// TwinCAT 3 PLC project PLC
// ProgramVersion: 3.1.4023.0
// libraries:
//   Tc2_Standard, * (Beckhoff Automation GmbH)
//   Tc2_System, * (Beckhoff Automation GmbH)
//   Tc3_Module, * (Beckhoff Automation GmbH)
// project tree:
//   / PlcTask.TcTTO
//   POUs/ MAIN.TcPOU
//   DUTs/IO/PDOs/ InfoData_6F19DB2B.TcDUT, YVR_Inputs_4719D0DB.TcDUT, YVR_Outputs_31F2CBB3.TcDUT, WcState_9091E0EB.TcDUT, InfoData_BEF6B88E.TcDUT, FB_Inputs_F0F03BDD.TcDUT, InfoData_A7436BC6.TcDUT, APS_Inputs_4719D0DB.TcDUT, APS_Diagdata_CE5B986F.TcDUT, APS_Comm_Inputs_388FE28E.TcDUT, APS_Outputs_31F2CBB3.TcDUT, APS_Comm_Outputs_082002A4.TcDUT, InfoData_E68C61CD.TcDUT, WcState_0B2B16F9.TcDUT, InfoData_2A97D6CF.TcDUT, Inputs_25A0042B.TcDUT, Outputs_2397A10E.TcDUT
//   DUTs/IO/Boxes/ EK1100_1FC0878B.TcDUT, EK1122_1FC0878B.TcDUT, APS1003_C6D7567B.TcDUT, APS1003_A49C5437.TcDUT, APS4322_7CC84994.TcDUT, APS4322_A49C5437.TcDUT
//   DUTs/IO/Devices/ SyncUnitTask_2D604ED5.TcDUT, SyncUnitTasks_6FEB8257.TcDUT, SyncUnits_99E584AF.TcDUT
//   DUTs/IO/Topology/ Beckhoff_APS1xxxEK1122_94631AF6.TcDUT, Beckhoff_APS1xxx_5C0D85AF.TcDUT, Beckhoff_APS4xxxEK1122_0B49C1F2.TcDUT, Beckhoff_APS4xxx_9BEEA20F.TcDUT, EtherCAT_Master_APSxxxx_214E63DA.TcDUT
//   DUTs/IO/Base/ EtcSlaveBase_82538BE2.TcDUT, EtcSlaveBase_82538BE2.TcDUT, EtcSlaveBase_82538BE2.TcDUT, EtcSlaveTerminalBase_947E5A46.TcDUT, EtcSlaveBoxBase_77A0E4A7.TcDUT, EtcSlaveEndTerminalBase_866C7F0C.TcDUT, InputBase_8311D824.TcDUT, OutputBase_10CEE7DE.TcDUT, EtcMasterBase_62654B43.TcDUT
//   GVLs/ GVL_iXlinker.TcGVL
// real-time tasks:
//   TASK PlcTask: cycle T#10ms, priority 20, ADS port 350
// I/O:
//   DEVICE EtherCAT_Master_APSxxxx, AmsNetId 172.20.30.238.3.1
//     Beckhoff APS1xxx [EK1100 EtherCAT Coupler (2A E-Bus)]
//       Beckhoff APS1xxxEK1122 [EK1122 2 port EtherCAT junction]
//         Beckhoff APS1xxxsub EK1100 [EK1100 EtherCAT Coupler (2A E-Bus)]
//         A_0001(APS1003-7000-0016) [APS1003-7000 Drive]
//       A_0002(APS1003-5000-0016) [APS1003-5000 Feedback]
//     Beckhoff APS4xxx [EK1100 EtherCAT Coupler (2A E-Bus)]
//       Beckhoff APS4xxxEK1122 [EK1122 2 port EtherCAT junction]
//         Beckhoff APS4xxxsub EK1100 [EK1100 EtherCAT Coupler (2A E-Bus)]
//         A_0001(APS4322-7000-0017) [APS4322-7000 Drive]
//       A_0002(APS4322-5000-0017) [APS4322-5000 Feedback]
// variable links:
//   PLC/PLC Instance <-> EtherCAT Master APSxxxx/Beckhoff APS1xxx
//     PlcTask Inputs/GVL_iXlinker.EtherCAT_Master_APSxxxx.Beckhoff_APS1xxx.InfoData.State <-> InfoData/State
//   PLC/PLC Instance <-> EtherCAT Master APSxxxx/Beckhoff APS1xxx/Beckhoff APS1xxxEK1122
//     PlcTask Inputs/GVL_iXlinker.EtherCAT_Master_APSxxxx.Beckhoff_APS1xxx.Beckhoff_APS1xxxEK1122.InfoData.State <-> InfoData/State
//   PLC/PLC Instance <-> EtherCAT Master APSxxxx/Beckhoff APS1xxx/Beckhoff APS1xxxEK1122/Beckhoff APS1xxxsub EK1100
//     PlcTask Inputs/GVL_iXlinker.EtherCAT_Master_APSxxxx.Beckhoff_APS1xxx.Beckhoff_APS1xxxEK1122.Beckhoff_APS1xxxsub_EK1100.InfoData.State <-> InfoData/State
//   PLC/PLC Instance <-> EtherCAT Master APSxxxx/Beckhoff APS1xxx/Beckhoff APS1xxxEK1122/A_0001(APS1003-7000-0016)
//     PlcTask Inputs/GVL_iXlinker.EtherCAT_Master_APSxxxx.Beckhoff_APS1xxx.Beckhoff_APS1xxxEK1122.A_0001_APS1003_7000_0016.YVR_Inputs.StatusWord <-> YVR Inputs/StatusWord
//     PlcTask Inputs/GVL_iXlinker.EtherCAT_Master_APSxxxx.Beckhoff_APS1xxx.Beckhoff_APS1xxxEK1122.A_0001_APS1003_7000_0016.YVR_Inputs.Current_D_0X0 <-> YVR Inputs/Current D 0X0
//     PlcTask Inputs/GVL_iXlinker.EtherCAT_Master_APSxxxx.Beckhoff_APS1xxx.Beckhoff_APS1xxxEK1122.A_0001_APS1003_7000_0016.YVR_Inputs.Current_D_0X1 <-> YVR Inputs/Current D 0X1
//     PlcTask Inputs/GVL_iXlinker.EtherCAT_Master_APSxxxx.Beckhoff_APS1xxx.Beckhoff_APS1xxxEK1122.A_0001_APS1003_7000_0016.YVR_Inputs.Current_D_0X2 <-> YVR Inputs/Current D 0X2
//     PlcTask Inputs/GVL_iXlinker.EtherCAT_Master_APSxxxx.Beckhoff_APS1xxx.Beckhoff_APS1xxxEK1122.A_0001_APS1003_7000_0016.YVR_Inputs.Current_D_1X0 <-> YVR Inputs/Current D 1X0
//     PlcTask Inputs/GVL_iXlinker.EtherCAT_Master_APSxxxx.Beckhoff_APS1xxx.Beckhoff_APS1xxxEK1122.A_0001_APS1003_7000_0016.YVR_Inputs.Current_D_1X1 <-> YVR Inputs/Current D 1X1
//     PlcTask Inputs/GVL_iXlinker.EtherCAT_Master_APSxxxx.Beckhoff_APS1xxx.Beckhoff_APS1xxxEK1122.A_0001_APS1003_7000_0016.YVR_Inputs.Current_D_1X2 <-> YVR Inputs/Current D 1X2
//     PlcTask Inputs/GVL_iXlinker.EtherCAT_Master_APSxxxx.Beckhoff_APS1xxx.Beckhoff_APS1xxxEK1122.A_0001_APS1003_7000_0016.YVR_Inputs.Current_D_2X0 <-> YVR Inputs/Current D 2X0
//     PlcTask Inputs/GVL_iXlinker.EtherCAT_Master_APSxxxx.Beckhoff_APS1xxx.Beckhoff_APS1xxxEK1122.A_0001_APS1003_7000_0016.YVR_Inputs.Current_D_2X1 <-> YVR Inputs/Current D 2X1
//     PlcTask Inputs/GVL_iXlinker.EtherCAT_Master_APSxxxx.Beckhoff_APS1xxx.Beckhoff_APS1xxxEK1122.A_0001_APS1003_7000_0016.YVR_Inputs.Current_D_2X2 <-> YVR Inputs/Current D 2X2
//     PlcTask Inputs/GVL_iXlinker.EtherCAT_Master_APSxxxx.Beckhoff_APS1xxx.Beckhoff_APS1xxxEK1122.A_0001_APS1003_7000_0016.YVR_Inputs.Current_D_3X0 <-> YVR Inputs/Current D 3X0
//     PlcTask Inputs/GVL_iXlinker.EtherCAT_Master_APSxxxx.Beckhoff_APS1xxx.Beckhoff_APS1xxxEK1122.A_0001_APS1003_7000_0016.YVR_Inputs.Current_D_3X1 <-> YVR Inputs/Current D 3X1
//     PlcTask Inputs/GVL_iXlinker.EtherCAT_Master_APSxxxx.Beckhoff_APS1xxx.Beckhoff_APS1xxxEK1122.A_0001_APS1003_7000_0016.YVR_Inputs.Current_D_3X2 <-> YVR Inputs/Current D 3X2
//     PlcTask Inputs/GVL_iXlinker.EtherCAT_Master_APSxxxx.Beckhoff_APS1xxx.Beckhoff_APS1xxxEK1122.A_0001_APS1003_7000_0016.YVR_Inputs.Current_D_0Y0 <-> YVR Inputs/Current D 0Y0
//     PlcTask Inputs/GVL_iXlinker.EtherCAT_Master_APSxxxx.Beckhoff_APS1xxx.Beckhoff_APS1xxxEK1122.A_0001_APS1003_7000_0016.YVR_Inputs.Current_D_0Y1 <-> YVR Inputs/Current D 0Y1
//     PlcTask Inputs/GVL_iXlinker.EtherCAT_Master_APSxxxx.Beckhoff_APS1xxx.Beckhoff_APS1xxxEK1122.A_0001_APS1003_7000_0016.YVR_Inputs.Current_D_0Y2 <-> YVR Inputs/Current D 0Y2
//     PlcTask Inputs/GVL_iXlinker.EtherCAT_Master_APSxxxx.Beckhoff_APS1xxx.Beckhoff_APS1xxxEK1122.A_0001_APS1003_7000_0016.YVR_Inputs.Current_D_1Y0 <-> YVR Inputs/Current D 1Y0
//     PlcTask Inputs/GVL_iXlinker.EtherCAT_Master_APSxxxx.Beckhoff_APS1xxx.Beckhoff_APS1xxxEK1122.A_0001_APS1003_7000_0016.YVR_Inputs.Current_D_1Y1 <-> YVR Inputs/Current D 1Y1
//     PlcTask Inputs/GVL_iXlinker.EtherCAT_Master_APSxxxx.Beckhoff_APS1xxx.Beckhoff_APS1xxxEK1122.A_0001_APS1003_7000_0016.YVR_Inputs.Current_D_1Y2 <-> YVR Inputs/Current D 1Y2
//     PlcTask Inputs/GVL_iXlinker.EtherCAT_Master_APSxxxx.Beckhoff_APS1xxx.Beckhoff_APS1xxxEK1122.A_0001_APS1003_7000_0016.YVR_Inputs.Current_D_2Y0 <-> YVR Inputs/Current D 2Y0
//     PlcTask Inputs/GVL_iXlinker.EtherCAT_Master_APSxxxx.Beckhoff_APS1xxx.Beckhoff_APS1xxxEK1122.A_0001_APS1003_7000_0016.YVR_Inputs.Current_D_2Y1 <-> YVR Inputs/Current D 2Y1
//     PlcTask Inputs/GVL_iXlinker.EtherCAT_Master_APSxxxx.Beckhoff_APS1xxx.Beckhoff_APS1xxxEK1122.A_0001_APS1003_7000_0016.YVR_Inputs.Current_D_2Y2 <-> YVR Inputs/Current D 2Y2
//     PlcTask Inputs/GVL_iXlinker.EtherCAT_Master_APSxxxx.Beckhoff_APS1xxx.Beckhoff_APS1xxxEK1122.A_0001_APS1003_7000_0016.YVR_Inputs.Current_D_3Y0 <-> YVR Inputs/Current D 3Y0
//     PlcTask Inputs/GVL_iXlinker.EtherCAT_Master_APSxxxx.Beckhoff_APS1xxx.Beckhoff_APS1xxxEK1122.A_0001_APS1003_7000_0016.YVR_Inputs.Current_D_3Y1 <-> YVR Inputs/Current D 3Y1
//     PlcTask Inputs/GVL_iXlinker.EtherCAT_Master_APSxxxx.Beckhoff_APS1xxx.Beckhoff_APS1xxxEK1122.A_0001_APS1003_7000_0016.YVR_Inputs.Current_D_3Y2 <-> YVR Inputs/Current D 3Y2
//     PlcTask Inputs/GVL_iXlinker.EtherCAT_Master_APSxxxx.Beckhoff_APS1xxx.Beckhoff_APS1xxxEK1122.A_0001_APS1003_7000_0016.YVR_Inputs.Current_Q_0X0 <-> YVR Inputs/Current Q 0X0
//     PlcTask Inputs/GVL_iXlinker.EtherCAT_Master_APSxxxx.Beckhoff_APS1xxx.Beckhoff_APS1xxxEK1122.A_0001_APS1003_7000_0016.YVR_Inputs.Current_Q_0X1 <-> YVR Inputs/Current Q 0X1
//     PlcTask Inputs/GVL_iXlinker.EtherCAT_Master_APSxxxx.Beckhoff_APS1xxx.Beckhoff_APS1xxxEK1122.A_0001_APS1003_7000_0016.YVR_Inputs.Current_Q_0X2 <-> YVR Inputs/Current Q 0X2
//     PlcTask Inputs/GVL_iXlinker.EtherCAT_Master_APSxxxx.Beckhoff_APS1xxx.Beckhoff_APS1xxxEK1122.A_0001_APS1003_7000_0016.YVR_Inputs.Current_Q_1X0 <-> YVR Inputs/Current Q 1X0
//     PlcTask Inputs/GVL_iXlinker.EtherCAT_Master_APSxxxx.Beckhoff_APS1xxx.Beckhoff_APS1xxxEK1122.A_0001_APS1003_7000_0016.YVR_Inputs.Current_Q_1X1 <-> YVR Inputs/Current Q 1X1
//     PlcTask Inputs/GVL_iXlinker.EtherCAT_Master_APSxxxx.Beckhoff_APS1xxx.Beckhoff_APS1xxxEK1122.A_0001_APS1003_7000_0016.YVR_Inputs.Current_Q_1X2 <-> YVR Inputs/Current Q 1X2
//     PlcTask Inputs/GVL_iXlinker.EtherCAT_Master_APSxxxx.Beckhoff_APS1xxx.Beckhoff_APS1xxxEK1122.A_0001_APS1003_7000_0016.YVR_Inputs.Current_Q_2X0 <-> YVR Inputs/Current Q 2X0
//     PlcTask Inputs/GVL_iXlinker.EtherCAT_Master_APSxxxx.Beckhoff_APS1xxx.Beckhoff_APS1xxxEK1122.A_0001_APS1003_7000_0016.YVR_Inputs.Current_Q_2X1 <-> YVR Inputs/Current Q 2X1
//     PlcTask Inputs/GVL_iXlinker.EtherCAT_Master_APSxxxx.Beckhoff_APS1xxx.Beckhoff_APS1xxxEK1122.A_0001_APS1003_7000_0016.YVR_Inputs.Current_Q_2X2 <-> YVR Inputs/Current Q 2X2
//     PlcTask Inputs/GVL_iXlinker.EtherCAT_Master_APSxxxx.Beckhoff_APS1xxx.Beckhoff_APS1xxxEK1122.A_0001_APS1003_7000_0016.YVR_Inputs.Current_Q_3X0 <-> YVR Inputs/Current Q 3X0
//     PlcTask Inputs/GVL_iXlinker.EtherCAT_Master_APSxxxx.Beckhoff_APS1xxx.Beckhoff_APS1xxxEK1122.A_0001_APS1003_7000_0016.YVR_Inputs.Current_Q_3X1 <-> YVR Inputs/Current Q 3X1
//     PlcTask Inputs/GVL_iXlinker.EtherCAT_Master_APSxxxx.Beckhoff_APS1xxx.Beckhoff_APS1xxxEK1122.A_0001_APS1003_7000_0016.YVR_Inputs.Current_Q_3X2 <-> YVR Inputs/Current Q 3X2
//     PlcTask Inputs/GVL_iXlinker.EtherCAT_Master_APSxxxx.Beckhoff_APS1xxx.Beckhoff_APS1xxxEK1122.A_0001_APS1003_7000_0016.YVR_Inputs.Current_Q_0Y0 <-> YVR Inputs/Current Q 0Y0
//     PlcTask Inputs/GVL_iXlinker.EtherCAT_Master_APSxxxx.Beckhoff_APS1xxx.Beckhoff_APS1xxxEK1122.A_0001_APS1003_7000_0016.YVR_Inputs.Current_Q_0Y1 <-> YVR Inputs/Current Q 0Y1
//     PlcTask Inputs/GVL_iXlinker.EtherCAT_Master_APSxxxx.Beckhoff_APS1xxx.Beckhoff_APS1xxxEK1122.A_0001_APS1003_7000_0016.YVR_Inputs.Current_Q_0Y2 <-> YVR Inputs/Current Q 0Y2
//     PlcTask Inputs/GVL_iXlinker.EtherCAT_Master_APSxxxx.Beckhoff_APS1xxx.Beckhoff_APS1xxxEK1122.A_0001_APS1003_7000_0016.YVR_Inputs.Current_Q_1Y0 <-> YVR Inputs/Current Q 1Y0
//     PlcTask Inputs/GVL_iXlinker.EtherCAT_Master_APSxxxx.Beckhoff_APS1xxx.Beckhoff_APS1xxxEK1122.A_0001_APS1003_7000_0016.YVR_Inputs.Current_Q_1Y1 <-> YVR Inputs/Current Q 1Y1
//     PlcTask Inputs/GVL_iXlinker.EtherCAT_Master_APSxxxx.Beckhoff_APS1xxx.Beckhoff_APS1xxxEK1122.A_0001_APS1003_7000_0016.YVR_Inputs.Current_Q_1Y2 <-> YVR Inputs/Current Q 1Y2
//     PlcTask Inputs/GVL_iXlinker.EtherCAT_Master_APSxxxx.Beckhoff_APS1xxx.Beckhoff_APS1xxxEK1122.A_0001_APS1003_7000_0016.YVR_Inputs.Current_Q_2Y0 <-> YVR Inputs/Current Q 2Y0
//     PlcTask Inputs/GVL_iXlinker.EtherCAT_Master_APSxxxx.Beckhoff_APS1xxx.Beckhoff_APS1xxxEK1122.A_0001_APS1003_7000_0016.YVR_Inputs.Current_Q_2Y1 <-> YVR Inputs/Current Q 2Y1
//     PlcTask Inputs/GVL_iXlinker.EtherCAT_Master_APSxxxx.Beckhoff_APS1xxx.Beckhoff_APS1xxxEK1122.A_0001_APS1003_7000_0016.YVR_Inputs.Current_Q_2Y2 <-> YVR Inputs/Current Q 2Y2
//     PlcTask Inputs/GVL_iXlinker.EtherCAT_Master_APSxxxx.Beckhoff_APS1xxx.Beckhoff_APS1xxxEK1122.A_0001_APS1003_7000_0016.YVR_Inputs.Current_Q_3Y0 <-> YVR Inputs/Current Q 3Y0
//     PlcTask Inputs/GVL_iXlinker.EtherCAT_Master_APSxxxx.Beckhoff_APS1xxx.Beckhoff_APS1xxxEK1122.A_0001_APS1003_7000_0016.YVR_Inputs.Current_Q_3Y1 <-> YVR Inputs/Current Q 3Y1
//     PlcTask Inputs/GVL_iXlinker.EtherCAT_Master_APSxxxx.Beckhoff_APS1xxx.Beckhoff_APS1xxxEK1122.A_0001_APS1003_7000_0016.YVR_Inputs.Current_Q_3Y2 <-> YVR Inputs/Current Q 3Y2
//     PlcTask Outputs/GVL_iXlinker.EtherCAT_Master_APSxxxx.Beckhoff_APS1xxx.Beckhoff_APS1xxxEK1122.A_0001_APS1003_7000_0016.YVR_Outputs.ControlWord <-> YVR Outputs/ControlWord
//     PlcTask Outputs/GVL_iXlinker.EtherCAT_Master_APSxxxx.Beckhoff_APS1xxx.Beckhoff_APS1xxxEK1122.A_0001_APS1003_7000_0016.YVR_Outputs.Current_D_0X0 <-> YVR Outputs/Current D 0X0
//     PlcTask Outputs/GVL_iXlinker.EtherCAT_Master_APSxxxx.Beckhoff_APS1xxx.Beckhoff_APS1xxxEK1122.A_0001_APS1003_7000_0016.YVR_Outputs.Current_D_0X1 <-> YVR Outputs/Current D 0X1
//     PlcTask Outputs/GVL_iXlinker.EtherCAT_Master_APSxxxx.Beckhoff_APS1xxx.Beckhoff_APS1xxxEK1122.A_0001_APS1003_7000_0016.YVR_Outputs.Current_D_0X2 <-> YVR Outputs/Current D 0X2
//     PlcTask Outputs/GVL_iXlinker.EtherCAT_Master_APSxxxx.Beckhoff_APS1xxx.Beckhoff_APS1xxxEK1122.A_0001_APS1003_7000_0016.YVR_Outputs.Current_D_1X0 <-> YVR Outputs/Current D 1X0
//     PlcTask Outputs/GVL_iXlinker.EtherCAT_Master_APSxxxx.Beckhoff_APS1xxx.Beckhoff_APS1xxxEK1122.A_0001_APS1003_7000_0016.YVR_Outputs.Current_D_1X1 <-> YVR Outputs/Current D 1X1
//     PlcTask Outputs/GVL_iXlinker.EtherCAT_Master_APSxxxx.Beckhoff_APS1xxx.Beckhoff_APS1xxxEK1122.A_0001_APS1003_7000_0016.YVR_Outputs.Current_D_1X2 <-> YVR Outputs/Current D 1X2
//     PlcTask Outputs/GVL_iXlinker.EtherCAT_Master_APSxxxx.Beckhoff_APS1xxx.Beckhoff_APS1xxxEK1122.A_0001_APS1003_7000_0016.YVR_Outputs.Current_D_2X0 <-> YVR Outputs/Current D 2X0
//     PlcTask Outputs/GVL_iXlinker.EtherCAT_Master_APSxxxx.Beckhoff_APS1xxx.Beckhoff_APS1xxxEK1122.A_0001_APS1003_7000_0016.YVR_Outputs.Current_D_2X1 <-> YVR Outputs/Current D 2X1
//     PlcTask Outputs/GVL_iXlinker.EtherCAT_Master_APSxxxx.Beckhoff_APS1xxx.Beckhoff_APS1xxxEK1122.A_0001_APS1003_7000_0016.YVR_Outputs.Current_D_2X2 <-> YVR Outputs/Current D 2X2
//     PlcTask Outputs/GVL_iXlinker.EtherCAT_Master_APSxxxx.Beckhoff_APS1xxx.Beckhoff_APS1xxxEK1122.A_0001_APS1003_7000_0016.YVR_Outputs.Current_D_3X0 <-> YVR Outputs/Current D 3X0
//     PlcTask Outputs/GVL_iXlinker.EtherCAT_Master_APSxxxx.Beckhoff_APS1xxx.Beckhoff_APS1xxxEK1122.A_0001_APS1003_7000_0016.YVR_Outputs.Current_D_3X1 <-> YVR Outputs/Current D 3X1
//     PlcTask Outputs/GVL_iXlinker.EtherCAT_Master_APSxxxx.Beckhoff_APS1xxx.Beckhoff_APS1xxxEK1122.A_0001_APS1003_7000_0016.YVR_Outputs.Current_D_3X2 <-> YVR Outputs/Current D 3X2
//     PlcTask Outputs/GVL_iXlinker.EtherCAT_Master_APSxxxx.Beckhoff_APS1xxx.Beckhoff_APS1xxxEK1122.A_0001_APS1003_7000_0016.YVR_Outputs.Current_D_0Y0 <-> YVR Outputs/Current D 0Y0
//     PlcTask Outputs/GVL_iXlinker.EtherCAT_Master_APSxxxx.Beckhoff_APS1xxx.Beckhoff_APS1xxxEK1122.A_0001_APS1003_7000_0016.YVR_Outputs.Current_D_0Y1 <-> YVR Outputs/Current D 0Y1
//     PlcTask Outputs/GVL_iXlinker.EtherCAT_Master_APSxxxx.Beckhoff_APS1xxx.Beckhoff_APS1xxxEK1122.A_0001_APS1003_7000_0016.YVR_Outputs.Current_D_0Y2 <-> YVR Outputs/Current D 0Y2
//     PlcTask Outputs/GVL_iXlinker.EtherCAT_Master_APSxxxx.Beckhoff_APS1xxx.Beckhoff_APS1xxxEK1122.A_0001_APS1003_7000_0016.YVR_Outputs.Current_D_1Y0 <-> YVR Outputs/Current D 1Y0
//     PlcTask Outputs/GVL_iXlinker.EtherCAT_Master_APSxxxx.Beckhoff_APS1xxx.Beckhoff_APS1xxxEK1122.A_0001_APS1003_7000_0016.YVR_Outputs.Current_D_1Y1 <-> YVR Outputs/Current D 1Y1
//     PlcTask Outputs/GVL_iXlinker.EtherCAT_Master_APSxxxx.Beckhoff_APS1xxx.Beckhoff_APS1xxxEK1122.A_0001_APS1003_7000_0016.YVR_Outputs.Current_D_1Y2 <-> YVR Outputs/Current D 1Y2
//     PlcTask Outputs/GVL_iXlinker.EtherCAT_Master_APSxxxx.Beckhoff_APS1xxx.Beckhoff_APS1xxxEK1122.A_0001_APS1003_7000_0016.YVR_Outputs.Current_D_2Y0 <-> YVR Outputs/Current D 2Y0
//     PlcTask Outputs/GVL_iXlinker.EtherCAT_Master_APSxxxx.Beckhoff_APS1xxx.Beckhoff_APS1xxxEK1122.A_0001_APS1003_7000_0016.YVR_Outputs.Current_D_2Y1 <-> YVR Outputs/Current D 2Y1
//     PlcTask Outputs/GVL_iXlinker.EtherCAT_Master_APSxxxx.Beckhoff_APS1xxx.Beckhoff_APS1xxxEK1122.A_0001_APS1003_7000_0016.YVR_Outputs.Current_D_2Y2 <-> YVR Outputs/Current D 2Y2
//     PlcTask Outputs/GVL_iXlinker.EtherCAT_Master_APSxxxx.Beckhoff_APS1xxx.Beckhoff_APS1xxxEK1122.A_0001_APS1003_7000_0016.YVR_Outputs.Current_D_3Y0 <-> YVR Outputs/Current D 3Y0
//     PlcTask Outputs/GVL_iXlinker.EtherCAT_Master_APSxxxx.Beckhoff_APS1xxx.Beckhoff_APS1xxxEK1122.A_0001_APS1003_7000_0016.YVR_Outputs.Current_D_3Y1 <-> YVR Outputs/Current D 3Y1
//     PlcTask Outputs/GVL_iXlinker.EtherCAT_Master_APSxxxx.Beckhoff_APS1xxx.Beckhoff_APS1xxxEK1122.A_0001_APS1003_7000_0016.YVR_Outputs.Current_D_3Y2 <-> YVR Outputs/Current D 3Y2
//     PlcTask Outputs/GVL_iXlinker.EtherCAT_Master_APSxxxx.Beckhoff_APS1xxx.Beckhoff_APS1xxxEK1122.A_0001_APS1003_7000_0016.YVR_Outputs.Current_Q_0X0 <-> YVR Outputs/Current Q 0X0
//     PlcTask Outputs/GVL_iXlinker.EtherCAT_Master_APSxxxx.Beckhoff_APS1xxx.Beckhoff_APS1xxxEK1122.A_0001_APS1003_7000_0016.YVR_Outputs.Current_Q_0X1 <-> YVR Outputs/Current Q 0X1
//     PlcTask Outputs/GVL_iXlinker.EtherCAT_Master_APSxxxx.Beckhoff_APS1xxx.Beckhoff_APS1xxxEK1122.A_0001_APS1003_7000_0016.YVR_Outputs.Current_Q_0X2 <-> YVR Outputs/Current Q 0X2
//     PlcTask Outputs/GVL_iXlinker.EtherCAT_Master_APSxxxx.Beckhoff_APS1xxx.Beckhoff_APS1xxxEK1122.A_0001_APS1003_7000_0016.YVR_Outputs.Current_Q_1X0 <-> YVR Outputs/Current Q 1X0
//     PlcTask Outputs/GVL_iXlinker.EtherCAT_Master_APSxxxx.Beckhoff_APS1xxx.Beckhoff_APS1xxxEK1122.A_0001_APS1003_7000_0016.YVR_Outputs.Current_Q_1X1 <-> YVR Outputs/Current Q 1X1
//     PlcTask Outputs/GVL_iXlinker.EtherCAT_Master_APSxxxx.Beckhoff_APS1xxx.Beckhoff_APS1xxxEK1122.A_0001_APS1003_7000_0016.YVR_Outputs.Current_Q_1X2 <-> YVR Outputs/Current Q 1X2
//     PlcTask Outputs/GVL_iXlinker.EtherCAT_Master_APSxxxx.Beckhoff_APS1xxx.Beckhoff_APS1xxxEK1122.A_0001_APS1003_7000_0016.YVR_Outputs.Current_Q_2X0 <-> YVR Outputs/Current Q 2X0
//     PlcTask Outputs/GVL_iXlinker.EtherCAT_Master_APSxxxx.Beckhoff_APS1xxx.Beckhoff_APS1xxxEK1122.A_0001_APS1003_7000_0016.YVR_Outputs.Current_Q_2X1 <-> YVR Outputs/Current Q 2X1
//     PlcTask Outputs/GVL_iXlinker.EtherCAT_Master_APSxxxx.Beckhoff_APS1xxx.Beckhoff_APS1xxxEK1122.A_0001_APS1003_7000_0016.YVR_Outputs.Current_Q_2X2 <-> YVR Outputs/Current Q 2X2
//     PlcTask Outputs/GVL_iXlinker.EtherCAT_Master_APSxxxx.Beckhoff_APS1xxx.Beckhoff_APS1xxxEK1122.A_0001_APS1003_7000_0016.YVR_Outputs.Current_Q_3X0 <-> YVR Outputs/Current Q 3X0
//     PlcTask Outputs/GVL_iXlinker.EtherCAT_Master_APSxxxx.Beckhoff_APS1xxx.Beckhoff_APS1xxxEK1122.A_0001_APS1003_7000_0016.YVR_Outputs.Current_Q_3X1 <-> YVR Outputs/Current Q 3X1
//     PlcTask Outputs/GVL_iXlinker.EtherCAT_Master_APSxxxx.Beckhoff_APS1xxx.Beckhoff_APS1xxxEK1122.A_0001_APS1003_7000_0016.YVR_Outputs.Current_Q_3X2 <-> YVR Outputs/Current Q 3X2
//     PlcTask Outputs/GVL_iXlinker.EtherCAT_Master_APSxxxx.Beckhoff_APS1xxx.Beckhoff_APS1xxxEK1122.A_0001_APS1003_7000_0016.YVR_Outputs.Current_Q_0Y0 <-> YVR Outputs/Current Q 0Y0
//     PlcTask Outputs/GVL_iXlinker.EtherCAT_Master_APSxxxx.Beckhoff_APS1xxx.Beckhoff_APS1xxxEK1122.A_0001_APS1003_7000_0016.YVR_Outputs.Current_Q_0Y1 <-> YVR Outputs/Current Q 0Y1
//     PlcTask Outputs/GVL_iXlinker.EtherCAT_Master_APSxxxx.Beckhoff_APS1xxx.Beckhoff_APS1xxxEK1122.A_0001_APS1003_7000_0016.YVR_Outputs.Current_Q_0Y2 <-> YVR Outputs/Current Q 0Y2
//     PlcTask Outputs/GVL_iXlinker.EtherCAT_Master_APSxxxx.Beckhoff_APS1xxx.Beckhoff_APS1xxxEK1122.A_0001_APS1003_7000_0016.YVR_Outputs.Current_Q_1Y0 <-> YVR Outputs/Current Q 1Y0
//     PlcTask Outputs/GVL_iXlinker.EtherCAT_Master_APSxxxx.Beckhoff_APS1xxx.Beckhoff_APS1xxxEK1122.A_0001_APS1003_7000_0016.YVR_Outputs.Current_Q_1Y1 <-> YVR Outputs/Current Q 1Y1
//     PlcTask Outputs/GVL_iXlinker.EtherCAT_Master_APSxxxx.Beckhoff_APS1xxx.Beckhoff_APS1xxxEK1122.A_0001_APS1003_7000_0016.YVR_Outputs.Current_Q_1Y2 <-> YVR Outputs/Current Q 1Y2
//     PlcTask Outputs/GVL_iXlinker.EtherCAT_Master_APSxxxx.Beckhoff_APS1xxx.Beckhoff_APS1xxxEK1122.A_0001_APS1003_7000_0016.YVR_Outputs.Current_Q_2Y0 <-> YVR Outputs/Current Q 2Y0
//     PlcTask Outputs/GVL_iXlinker.EtherCAT_Master_APSxxxx.Beckhoff_APS1xxx.Beckhoff_APS1xxxEK1122.A_0001_APS1003_7000_0016.YVR_Outputs.Current_Q_2Y1 <-> YVR Outputs/Current Q 2Y1
//     PlcTask Outputs/GVL_iXlinker.EtherCAT_Master_APSxxxx.Beckhoff_APS1xxx.Beckhoff_APS1xxxEK1122.A_0001_APS1003_7000_0016.YVR_Outputs.Current_Q_2Y2 <-> YVR Outputs/Current Q 2Y2
//     PlcTask Outputs/GVL_iXlinker.EtherCAT_Master_APSxxxx.Beckhoff_APS1xxx.Beckhoff_APS1xxxEK1122.A_0001_APS1003_7000_0016.YVR_Outputs.Current_Q_3Y0 <-> YVR Outputs/Current Q 3Y0
//     PlcTask Outputs/GVL_iXlinker.EtherCAT_Master_APSxxxx.Beckhoff_APS1xxx.Beckhoff_APS1xxxEK1122.A_0001_APS1003_7000_0016.YVR_Outputs.Current_Q_3Y1 <-> YVR Outputs/Current Q 3Y1
//     PlcTask Outputs/GVL_iXlinker.EtherCAT_Master_APSxxxx.Beckhoff_APS1xxx.Beckhoff_APS1xxxEK1122.A_0001_APS1003_7000_0016.YVR_Outputs.Current_Q_3Y2 <-> YVR Outputs/Current Q 3Y2
//     PlcTask Outputs/GVL_iXlinker.EtherCAT_Master_APSxxxx.Beckhoff_APS1xxx.Beckhoff_APS1xxxEK1122.A_0001_APS1003_7000_0016.YVR_Outputs.PhiE_0X0 <-> YVR Outputs/PhiE 0X0
//     PlcTask Outputs/GVL_iXlinker.EtherCAT_Master_APSxxxx.Beckhoff_APS1xxx.Beckhoff_APS1xxxEK1122.A_0001_APS1003_7000_0016.YVR_Outputs.PhiE_0X1 <-> YVR Outputs/PhiE 0X1
//     PlcTask Outputs/GVL_iXlinker.EtherCAT_Master_APSxxxx.Beckhoff_APS1xxx.Beckhoff_APS1xxxEK1122.A_0001_APS1003_7000_0016.YVR_Outputs.PhiE_0X2 <-> YVR Outputs/PhiE 0X2
//     PlcTask Outputs/GVL_iXlinker.EtherCAT_Master_APSxxxx.Beckhoff_APS1xxx.Beckhoff_APS1xxxEK1122.A_0001_APS1003_7000_0016.YVR_Outputs.PhiE_1X0 <-> YVR Outputs/PhiE 1X0
//     PlcTask Outputs/GVL_iXlinker.EtherCAT_Master_APSxxxx.Beckhoff_APS1xxx.Beckhoff_APS1xxxEK1122.A_0001_APS1003_7000_0016.YVR_Outputs.PhiE_1X1 <-> YVR Outputs/PhiE 1X1
//     PlcTask Outputs/GVL_iXlinker.EtherCAT_Master_APSxxxx.Beckhoff_APS1xxx.Beckhoff_APS1xxxEK1122.A_0001_APS1003_7000_0016.YVR_Outputs.PhiE_1X2 <-> YVR Outputs/PhiE 1X2
//     PlcTask Outputs/GVL_iXlinker.EtherCAT_Master_APSxxxx.Beckhoff_APS1xxx.Beckhoff_APS1xxxEK1122.A_0001_APS1003_7000_0016.YVR_Outputs.PhiE_2X0 <-> YVR Outputs/PhiE 2X0
//     PlcTask Outputs/GVL_iXlinker.EtherCAT_Master_APSxxxx.Beckhoff_APS1xxx.Beckhoff_APS1xxxEK1122.A_0001_APS1003_7000_0016.YVR_Outputs.PhiE_2X1 <-> YVR Outputs/PhiE 2X1
//     PlcTask Outputs/GVL_iXlinker.EtherCAT_Master_APSxxxx.Beckhoff_APS1xxx.Beckhoff_APS1xxxEK1122.A_0001_APS1003_7000_0016.YVR_Outputs.PhiE_2X2 <-> YVR Outputs/PhiE 2X2
//     PlcTask Outputs/GVL_iXlinker.EtherCAT_Master_APSxxxx.Beckhoff_APS1xxx.Beckhoff_APS1xxxEK1122.A_0001_APS1003_7000_0016.YVR_Outputs.PhiE_3X0 <-> YVR Outputs/PhiE 3X0
//     PlcTask Outputs/GVL_iXlinker.EtherCAT_Master_APSxxxx.Beckhoff_APS1xxx.Beckhoff_APS1xxxEK1122.A_0001_APS1003_7000_0016.YVR_Outputs.PhiE_3X1 <-> YVR Outputs/PhiE 3X1
//     PlcTask Outputs/GVL_iXlinker.EtherCAT_Master_APSxxxx.Beckhoff_APS1xxx.Beckhoff_APS1xxxEK1122.A_0001_APS1003_7000_0016.YVR_Outputs.PhiE_3X2 <-> YVR Outputs/PhiE 3X2
//     PlcTask Outputs/GVL_iXlinker.EtherCAT_Master_APSxxxx.Beckhoff_APS1xxx.Beckhoff_APS1xxxEK1122.A_0001_APS1003_7000_0016.YVR_Outputs.PhiE_0Y0 <-> YVR Outputs/PhiE 0Y0
//     PlcTask Outputs/GVL_iXlinker.EtherCAT_Master_APSxxxx.Beckhoff_APS1xxx.Beckhoff_APS1xxxEK1122.A_0001_APS1003_7000_0016.YVR_Outputs.PhiE_0Y1 <-> YVR Outputs/PhiE 0Y1
//     PlcTask Outputs/GVL_iXlinker.EtherCAT_Master_APSxxxx.Beckhoff_APS1xxx.Beckhoff_APS1xxxEK1122.A_0001_APS1003_7000_0016.YVR_Outputs.PhiE_0Y2 <-> YVR Outputs/PhiE 0Y2
//     PlcTask Outputs/GVL_iXlinker.EtherCAT_Master_APSxxxx.Beckhoff_APS1xxx.Beckhoff_APS1xxxEK1122.A_0001_APS1003_7000_0016.YVR_Outputs.PhiE_1Y0 <-> YVR Outputs/PhiE 1Y0
//     PlcTask Outputs/GVL_iXlinker.EtherCAT_Master_APSxxxx.Beckhoff_APS1xxx.Beckhoff_APS1xxxEK1122.A_0001_APS1003_7000_0016.YVR_Outputs.PhiE_1Y1 <-> YVR Outputs/PhiE 1Y1
//     PlcTask Outputs/GVL_iXlinker.EtherCAT_Master_APSxxxx.Beckhoff_APS1xxx.Beckhoff_APS1xxxEK1122.A_0001_APS1003_7000_0016.YVR_Outputs.PhiE_1Y2 <-> YVR Outputs/PhiE 1Y2
//     PlcTask Outputs/GVL_iXlinker.EtherCAT_Master_APSxxxx.Beckhoff_APS1xxx.Beckhoff_APS1xxxEK1122.A_0001_APS1003_7000_0016.YVR_Outputs.PhiE_2Y0 <-> YVR Outputs/PhiE 2Y0
//     PlcTask Outputs/GVL_iXlinker.EtherCAT_Master_APSxxxx.Beckhoff_APS1xxx.Beckhoff_APS1xxxEK1122.A_0001_APS1003_7000_0016.YVR_Outputs.PhiE_2Y1 <-> YVR Outputs/PhiE 2Y1
//     PlcTask Outputs/GVL_iXlinker.EtherCAT_Master_APSxxxx.Beckhoff_APS1xxx.Beckhoff_APS1xxxEK1122.A_0001_APS1003_7000_0016.YVR_Outputs.PhiE_2Y2 <-> YVR Outputs/PhiE 2Y2
//     PlcTask Outputs/GVL_iXlinker.EtherCAT_Master_APSxxxx.Beckhoff_APS1xxx.Beckhoff_APS1xxxEK1122.A_0001_APS1003_7000_0016.YVR_Outputs.PhiE_3Y0 <-> YVR Outputs/PhiE 3Y0
//     PlcTask Outputs/GVL_iXlinker.EtherCAT_Master_APSxxxx.Beckhoff_APS1xxx.Beckhoff_APS1xxxEK1122.A_0001_APS1003_7000_0016.YVR_Outputs.PhiE_3Y1 <-> YVR Outputs/PhiE 3Y1
//     PlcTask Outputs/GVL_iXlinker.EtherCAT_Master_APSxxxx.Beckhoff_APS1xxx.Beckhoff_APS1xxxEK1122.A_0001_APS1003_7000_0016.YVR_Outputs.PhiE_3Y2 <-> YVR Outputs/PhiE 3Y2
//     PlcTask Inputs/GVL_iXlinker.EtherCAT_Master_APSxxxx.Beckhoff_APS1xxx.Beckhoff_APS1xxxEK1122.A_0001_APS1003_7000_0016.WcState.WcState <-> WcState/WcState
//     PlcTask Inputs/GVL_iXlinker.EtherCAT_Master_APSxxxx.Beckhoff_APS1xxx.Beckhoff_APS1xxxEK1122.A_0001_APS1003_7000_0016.WcState.InputToggle <-> WcState/InputToggle
//     PlcTask Inputs/GVL_iXlinker.EtherCAT_Master_APSxxxx.Beckhoff_APS1xxx.Beckhoff_APS1xxxEK1122.A_0001_APS1003_7000_0016.InfoData.AdsAddr <-> InfoData/AdsAddr
//     PlcTask Inputs/GVL_iXlinker.EtherCAT_Master_APSxxxx.Beckhoff_APS1xxx.Beckhoff_APS1xxxEK1122.A_0001_APS1003_7000_0016.InfoData.DcOutputShift <-> InfoData/DcOutputShift
//     PlcTask Inputs/GVL_iXlinker.EtherCAT_Master_APSxxxx.Beckhoff_APS1xxx.Beckhoff_APS1xxxEK1122.A_0001_APS1003_7000_0016.InfoData.DcInputShift <-> InfoData/DcInputShift
//     PlcTask Inputs/GVL_iXlinker.EtherCAT_Master_APSxxxx.Beckhoff_APS1xxx.Beckhoff_APS1xxxEK1122.A_0001_APS1003_7000_0016.InfoData.State <-> InfoData/State
//   PLC/PLC Instance <-> EtherCAT Master APSxxxx/Beckhoff APS1xxx/A_0002(APS1003-5000-0016)
//     PlcTask Inputs/GVL_iXlinker.EtherCAT_Master_APSxxxx.Beckhoff_APS1xxx.A_0002_APS1003_5000_0016.FB_Inputs.Status <-> FB Inputs/Status
//     PlcTask Inputs/GVL_iXlinker.EtherCAT_Master_APSxxxx.Beckhoff_APS1xxx.A_0002_APS1003_5000_0016.FB_Inputs.A0_X_Field <-> FB Inputs/A0 X-Field
//     PlcTask Inputs/GVL_iXlinker.EtherCAT_Master_APSxxxx.Beckhoff_APS1xxx.A_0002_APS1003_5000_0016.FB_Inputs.A2_X_Field <-> FB Inputs/A2 X-Field
//     PlcTask Inputs/GVL_iXlinker.EtherCAT_Master_APSxxxx.Beckhoff_APS1xxx.A_0002_APS1003_5000_0016.FB_Inputs.A4_X_Field <-> FB Inputs/A4 X-Field
//     PlcTask Inputs/GVL_iXlinker.EtherCAT_Master_APSxxxx.Beckhoff_APS1xxx.A_0002_APS1003_5000_0016.FB_Inputs.A6_X_Field <-> FB Inputs/A6 X-Field
//     PlcTask Inputs/GVL_iXlinker.EtherCAT_Master_APSxxxx.Beckhoff_APS1xxx.A_0002_APS1003_5000_0016.FB_Inputs.A8_X_Field <-> FB Inputs/A8 X-Field
//     PlcTask Inputs/GVL_iXlinker.EtherCAT_Master_APSxxxx.Beckhoff_APS1xxx.A_0002_APS1003_5000_0016.FB_Inputs.A0_Y_Field <-> FB Inputs/A0 Y-Field
//     PlcTask Inputs/GVL_iXlinker.EtherCAT_Master_APSxxxx.Beckhoff_APS1xxx.A_0002_APS1003_5000_0016.FB_Inputs.A2_Y_Field <-> FB Inputs/A2 Y-Field
//     PlcTask Inputs/GVL_iXlinker.EtherCAT_Master_APSxxxx.Beckhoff_APS1xxx.A_0002_APS1003_5000_0016.FB_Inputs.A4_Y_Field <-> FB Inputs/A4 Y-Field
//     PlcTask Inputs/GVL_iXlinker.EtherCAT_Master_APSxxxx.Beckhoff_APS1xxx.A_0002_APS1003_5000_0016.FB_Inputs.A6_Y_Field <-> FB Inputs/A6 Y-Field
//     PlcTask Inputs/GVL_iXlinker.EtherCAT_Master_APSxxxx.Beckhoff_APS1xxx.A_0002_APS1003_5000_0016.FB_Inputs.A8_Y_Field <-> FB Inputs/A8 Y-Field
//     PlcTask Inputs/GVL_iXlinker.EtherCAT_Master_APSxxxx.Beckhoff_APS1xxx.A_0002_APS1003_5000_0016.FB_Inputs.A0_Z_Field <-> FB Inputs/A0 Z-Field
//     PlcTask Inputs/GVL_iXlinker.EtherCAT_Master_APSxxxx.Beckhoff_APS1xxx.A_0002_APS1003_5000_0016.FB_Inputs.A2_Z_Field <-> FB Inputs/A2 Z-Field
//     PlcTask Inputs/GVL_iXlinker.EtherCAT_Master_APSxxxx.Beckhoff_APS1xxx.A_0002_APS1003_5000_0016.FB_Inputs.A4_Z_Field <-> FB Inputs/A4 Z-Field
//     PlcTask Inputs/GVL_iXlinker.EtherCAT_Master_APSxxxx.Beckhoff_APS1xxx.A_0002_APS1003_5000_0016.FB_Inputs.A6_Z_Field <-> FB Inputs/A6 Z-Field
//     PlcTask Inputs/GVL_iXlinker.EtherCAT_Master_APSxxxx.Beckhoff_APS1xxx.A_0002_APS1003_5000_0016.FB_Inputs.A8_Z_Field <-> FB Inputs/A8 Z-Field
//     PlcTask Inputs/GVL_iXlinker.EtherCAT_Master_APSxxxx.Beckhoff_APS1xxx.A_0002_APS1003_5000_0016.FB_Inputs.B1_X_Field <-> FB Inputs/B1 X-Field
//     PlcTask Inputs/GVL_iXlinker.EtherCAT_Master_APSxxxx.Beckhoff_APS1xxx.A_0002_APS1003_5000_0016.FB_Inputs.B3_X_Field <-> FB Inputs/B3 X-Field
//     PlcTask Inputs/GVL_iXlinker.EtherCAT_Master_APSxxxx.Beckhoff_APS1xxx.A_0002_APS1003_5000_0016.FB_Inputs.B5_X_Field <-> FB Inputs/B5 X-Field
//     PlcTask Inputs/GVL_iXlinker.EtherCAT_Master_APSxxxx.Beckhoff_APS1xxx.A_0002_APS1003_5000_0016.FB_Inputs.B7_X_Field <-> FB Inputs/B7 X-Field
//     PlcTask Inputs/GVL_iXlinker.EtherCAT_Master_APSxxxx.Beckhoff_APS1xxx.A_0002_APS1003_5000_0016.FB_Inputs.B9_X_Field <-> FB Inputs/B9 X-Field
//     PlcTask Inputs/GVL_iXlinker.EtherCAT_Master_APSxxxx.Beckhoff_APS1xxx.A_0002_APS1003_5000_0016.FB_Inputs.B1_Y_Field <-> FB Inputs/B1 Y-Field
//     PlcTask Inputs/GVL_iXlinker.EtherCAT_Master_APSxxxx.Beckhoff_APS1xxx.A_0002_APS1003_5000_0016.FB_Inputs.B3_Y_Field <-> FB Inputs/B3 Y-Field
//     PlcTask Inputs/GVL_iXlinker.EtherCAT_Master_APSxxxx.Beckhoff_APS1xxx.A_0002_APS1003_5000_0016.FB_Inputs.B5_Y_Field <-> FB Inputs/B5 Y-Field
//     PlcTask Inputs/GVL_iXlinker.EtherCAT_Master_APSxxxx.Beckhoff_APS1xxx.A_0002_APS1003_5000_0016.FB_Inputs.B7_Y_Field <-> FB Inputs/B7 Y-Field
//     PlcTask Inputs/GVL_iXlinker.EtherCAT_Master_APSxxxx.Beckhoff_APS1xxx.A_0002_APS1003_5000_0016.FB_Inputs.B9_Y_Field <-> FB Inputs/B9 Y-Field
//     PlcTask Inputs/GVL_iXlinker.EtherCAT_Master_APSxxxx.Beckhoff_APS1xxx.A_0002_APS1003_5000_0016.FB_Inputs.B1_Z_Field <-> FB Inputs/B1 Z-Field
//     PlcTask Inputs/GVL_iXlinker.EtherCAT_Master_APSxxxx.Beckhoff_APS1xxx.A_0002_APS1003_5000_0016.FB_Inputs.B3_Z_Field <-> FB Inputs/B3 Z-Field
//     PlcTask Inputs/GVL_iXlinker.EtherCAT_Master_APSxxxx.Beckhoff_APS1xxx.A_0002_APS1003_5000_0016.FB_Inputs.B5_Z_Field <-> FB Inputs/B5 Z-Field
//     PlcTask Inputs/GVL_iXlinker.EtherCAT_Master_APSxxxx.Beckhoff_APS1xxx.A_0002_APS1003_5000_0016.FB_Inputs.B7_Z_Field <-> FB Inputs/B7 Z-Field
//     PlcTask Inputs/GVL_iXlinker.EtherCAT_Master_APSxxxx.Beckhoff_APS1xxx.A_0002_APS1003_5000_0016.FB_Inputs.B9_Z_Field <-> FB Inputs/B9 Z-Field
//     PlcTask Inputs/GVL_iXlinker.EtherCAT_Master_APSxxxx.Beckhoff_APS1xxx.A_0002_APS1003_5000_0016.FB_Inputs.C0_X_Field <-> FB Inputs/C0 X-Field
//     PlcTask Inputs/GVL_iXlinker.EtherCAT_Master_APSxxxx.Beckhoff_APS1xxx.A_0002_APS1003_5000_0016.FB_Inputs.C2_X_Field <-> FB Inputs/C2 X-Field
//     PlcTask Inputs/GVL_iXlinker.EtherCAT_Master_APSxxxx.Beckhoff_APS1xxx.A_0002_APS1003_5000_0016.FB_Inputs.C4_X_Field <-> FB Inputs/C4 X-Field
//     PlcTask Inputs/GVL_iXlinker.EtherCAT_Master_APSxxxx.Beckhoff_APS1xxx.A_0002_APS1003_5000_0016.FB_Inputs.C6_X_Field <-> FB Inputs/C6 X-Field
//     PlcTask Inputs/GVL_iXlinker.EtherCAT_Master_APSxxxx.Beckhoff_APS1xxx.A_0002_APS1003_5000_0016.FB_Inputs.C8_X_Field <-> FB Inputs/C8 X-Field
//     PlcTask Inputs/GVL_iXlinker.EtherCAT_Master_APSxxxx.Beckhoff_APS1xxx.A_0002_APS1003_5000_0016.FB_Inputs.C0_Y_Field <-> FB Inputs/C0 Y-Field
//     PlcTask Inputs/GVL_iXlinker.EtherCAT_Master_APSxxxx.Beckhoff_APS1xxx.A_0002_APS1003_5000_0016.FB_Inputs.C2_Y_Field <-> FB Inputs/C2 Y-Field
//     PlcTask Inputs/GVL_iXlinker.EtherCAT_Master_APSxxxx.Beckhoff_APS1xxx.A_0002_APS1003_5000_0016.FB_Inputs.C4_Y_Field <-> FB Inputs/C4 Y-Field
//     PlcTask Inputs/GVL_iXlinker.EtherCAT_Master_APSxxxx.Beckhoff_APS1xxx.A_0002_APS1003_5000_0016.FB_Inputs.C6_Y_Field <-> FB Inputs/C6 Y-Field
//     PlcTask Inputs/GVL_iXlinker.EtherCAT_Master_APSxxxx.Beckhoff_APS1xxx.A_0002_APS1003_5000_0016.FB_Inputs.C8_Y_Field <-> FB Inputs/C8 Y-Field
//     PlcTask Inputs/GVL_iXlinker.EtherCAT_Master_APSxxxx.Beckhoff_APS1xxx.A_0002_APS1003_5000_0016.FB_Inputs.C0_Z_Field <-> FB Inputs/C0 Z-Field
//     PlcTask Inputs/GVL_iXlinker.EtherCAT_Master_APSxxxx.Beckhoff_APS1xxx.A_0002_APS1003_5000_0016.FB_Inputs.C2_Z_Field <-> FB Inputs/C2 Z-Field
//     PlcTask Inputs/GVL_iXlinker.EtherCAT_Master_APSxxxx.Beckhoff_APS1xxx.A_0002_APS1003_5000_0016.FB_Inputs.C4_Z_Field <-> FB Inputs/C4 Z-Field
//     PlcTask Inputs/GVL_iXlinker.EtherCAT_Master_APSxxxx.Beckhoff_APS1xxx.A_0002_APS1003_5000_0016.FB_Inputs.C6_Z_Field <-> FB Inputs/C6 Z-Field
//     PlcTask Inputs/GVL_iXlinker.EtherCAT_Master_APSxxxx.Beckhoff_APS1xxx.A_0002_APS1003_5000_0016.FB_Inputs.C8_Z_Field <-> FB Inputs/C8 Z-Field
//     PlcTask Inputs/GVL_iXlinker.EtherCAT_Master_APSxxxx.Beckhoff_APS1xxx.A_0002_APS1003_5000_0016.FB_Inputs.D1_X_Field <-> FB Inputs/D1 X-Field
//     PlcTask Inputs/GVL_iXlinker.EtherCAT_Master_APSxxxx.Beckhoff_APS1xxx.A_0002_APS1003_5000_0016.FB_Inputs.D3_X_Field <-> FB Inputs/D3 X-Field
//     PlcTask Inputs/GVL_iXlinker.EtherCAT_Master_APSxxxx.Beckhoff_APS1xxx.A_0002_APS1003_5000_0016.FB_Inputs.D5_X_Field <-> FB Inputs/D5 X-Field
//     PlcTask Inputs/GVL_iXlinker.EtherCAT_Master_APSxxxx.Beckhoff_APS1xxx.A_0002_APS1003_5000_0016.FB_Inputs.D7_X_Field <-> FB Inputs/D7 X-Field
//     PlcTask Inputs/GVL_iXlinker.EtherCAT_Master_APSxxxx.Beckhoff_APS1xxx.A_0002_APS1003_5000_0016.FB_Inputs.D9_X_Field <-> FB Inputs/D9 X-Field
//     PlcTask Inputs/GVL_iXlinker.EtherCAT_Master_APSxxxx.Beckhoff_APS1xxx.A_0002_APS1003_5000_0016.FB_Inputs.D1_Y_Field <-> FB Inputs/D1 Y-Field
//     PlcTask Inputs/GVL_iXlinker.EtherCAT_Master_APSxxxx.Beckhoff_APS1xxx.A_0002_APS1003_5000_0016.FB_Inputs.D3_Y_Field <-> FB Inputs/D3 Y-Field
//     PlcTask Inputs/GVL_iXlinker.EtherCAT_Master_APSxxxx.Beckhoff_APS1xxx.A_0002_APS1003_5000_0016.FB_Inputs.D5_Y_Field <-> FB Inputs/D5 Y-Field
//     PlcTask Inputs/GVL_iXlinker.EtherCAT_Master_APSxxxx.Beckhoff_APS1xxx.A_0002_APS1003_5000_0016.FB_Inputs.D7_Y_Field <-> FB Inputs/D7 Y-Field
//     PlcTask Inputs/GVL_iXlinker.EtherCAT_Master_APSxxxx.Beckhoff_APS1xxx.A_0002_APS1003_5000_0016.FB_Inputs.D9_Y_Field <-> FB Inputs/D9 Y-Field
//     PlcTask Inputs/GVL_iXlinker.EtherCAT_Master_APSxxxx.Beckhoff_APS1xxx.A_0002_APS1003_5000_0016.FB_Inputs.D1_Z_Field <-> FB Inputs/D1 Z-Field
//     PlcTask Inputs/GVL_iXlinker.EtherCAT_Master_APSxxxx.Beckhoff_APS1xxx.A_0002_APS1003_5000_0016.FB_Inputs.D3_Z_Field <-> FB Inputs/D3 Z-Field
//     PlcTask Inputs/GVL_iXlinker.EtherCAT_Master_APSxxxx.Beckhoff_APS1xxx.A_0002_APS1003_5000_0016.FB_Inputs.D5_Z_Field <-> FB Inputs/D5 Z-Field
//     PlcTask Inputs/GVL_iXlinker.EtherCAT_Master_APSxxxx.Beckhoff_APS1xxx.A_0002_APS1003_5000_0016.FB_Inputs.D7_Z_Field <-> FB Inputs/D7 Z-Field
//     PlcTask Inputs/GVL_iXlinker.EtherCAT_Master_APSxxxx.Beckhoff_APS1xxx.A_0002_APS1003_5000_0016.FB_Inputs.D9_Z_Field <-> FB Inputs/D9 Z-Field
//     PlcTask Inputs/GVL_iXlinker.EtherCAT_Master_APSxxxx.Beckhoff_APS1xxx.A_0002_APS1003_5000_0016.FB_Inputs.E0_X_Field <-> FB Inputs/E0 X-Field
//     PlcTask Inputs/GVL_iXlinker.EtherCAT_Master_APSxxxx.Beckhoff_APS1xxx.A_0002_APS1003_5000_0016.FB_Inputs.E2_X_Field <-> FB Inputs/E2 X-Field
//     PlcTask Inputs/GVL_iXlinker.EtherCAT_Master_APSxxxx.Beckhoff_APS1xxx.A_0002_APS1003_5000_0016.FB_Inputs.E4_X_Field <-> FB Inputs/E4 X-Field
//     PlcTask Inputs/GVL_iXlinker.EtherCAT_Master_APSxxxx.Beckhoff_APS1xxx.A_0002_APS1003_5000_0016.FB_Inputs.E6_X_Field <-> FB Inputs/E6 X-Field
//     PlcTask Inputs/GVL_iXlinker.EtherCAT_Master_APSxxxx.Beckhoff_APS1xxx.A_0002_APS1003_5000_0016.FB_Inputs.E8_X_Field <-> FB Inputs/E8 X-Field
//     PlcTask Inputs/GVL_iXlinker.EtherCAT_Master_APSxxxx.Beckhoff_APS1xxx.A_0002_APS1003_5000_0016.FB_Inputs.E0_Y_Field <-> FB Inputs/E0 Y-Field
//     PlcTask Inputs/GVL_iXlinker.EtherCAT_Master_APSxxxx.Beckhoff_APS1xxx.A_0002_APS1003_5000_0016.FB_Inputs.E2_Y_Field <-> FB Inputs/E2 Y-Field
//     PlcTask Inputs/GVL_iXlinker.EtherCAT_Master_APSxxxx.Beckhoff_APS1xxx.A_0002_APS1003_5000_0016.FB_Inputs.E4_Y_Field <-> FB Inputs/E4 Y-Field
//     PlcTask Inputs/GVL_iXlinker.EtherCAT_Master_APSxxxx.Beckhoff_APS1xxx.A_0002_APS1003_5000_0016.FB_Inputs.E6_Y_Field <-> FB Inputs/E6 Y-Field
//     PlcTask Inputs/GVL_iXlinker.EtherCAT_Master_APSxxxx.Beckhoff_APS1xxx.A_0002_APS1003_5000_0016.FB_Inputs.E8_Y_Field <-> FB Inputs/E8 Y-Field
//     PlcTask Inputs/GVL_iXlinker.EtherCAT_Master_APSxxxx.Beckhoff_APS1xxx.A_0002_APS1003_5000_0016.FB_Inputs.E0_Z_Field <-> FB Inputs/E0 Z-Field
//     PlcTask Inputs/GVL_iXlinker.EtherCAT_Master_APSxxxx.Beckhoff_APS1xxx.A_0002_APS1003_5000_0016.FB_Inputs.E2_Z_Field <-> FB Inputs/E2 Z-Field
//     PlcTask Inputs/GVL_iXlinker.EtherCAT_Master_APSxxxx.Beckhoff_APS1xxx.A_0002_APS1003_5000_0016.FB_Inputs.E4_Z_Field <-> FB Inputs/E4 Z-Field
//     PlcTask Inputs/GVL_iXlinker.EtherCAT_Master_APSxxxx.Beckhoff_APS1xxx.A_0002_APS1003_5000_0016.FB_Inputs.E6_Z_Field <-> FB Inputs/E6 Z-Field
//     PlcTask Inputs/GVL_iXlinker.EtherCAT_Master_APSxxxx.Beckhoff_APS1xxx.A_0002_APS1003_5000_0016.FB_Inputs.E8_Z_Field <-> FB Inputs/E8 Z-Field
//     PlcTask Inputs/GVL_iXlinker.EtherCAT_Master_APSxxxx.Beckhoff_APS1xxx.A_0002_APS1003_5000_0016.FB_Inputs.F1_X_Field <-> FB Inputs/F1 X-Field
//     PlcTask Inputs/GVL_iXlinker.EtherCAT_Master_APSxxxx.Beckhoff_APS1xxx.A_0002_APS1003_5000_0016.FB_Inputs.F3_X_Field <-> FB Inputs/F3 X-Field
//     PlcTask Inputs/GVL_iXlinker.EtherCAT_Master_APSxxxx.Beckhoff_APS1xxx.A_0002_APS1003_5000_0016.FB_Inputs.F5_X_Field <-> FB Inputs/F5 X-Field
//     PlcTask Inputs/GVL_iXlinker.EtherCAT_Master_APSxxxx.Beckhoff_APS1xxx.A_0002_APS1003_5000_0016.FB_Inputs.F7_X_Field <-> FB Inputs/F7 X-Field
//     PlcTask Inputs/GVL_iXlinker.EtherCAT_Master_APSxxxx.Beckhoff_APS1xxx.A_0002_APS1003_5000_0016.FB_Inputs.F9_X_Field <-> FB Inputs/F9 X-Field
//     PlcTask Inputs/GVL_iXlinker.EtherCAT_Master_APSxxxx.Beckhoff_APS1xxx.A_0002_APS1003_5000_0016.FB_Inputs.F1_Y_Field <-> FB Inputs/F1 Y-Field
//     PlcTask Inputs/GVL_iXlinker.EtherCAT_Master_APSxxxx.Beckhoff_APS1xxx.A_0002_APS1003_5000_0016.FB_Inputs.F3_Y_Field <-> FB Inputs/F3 Y-Field
//     PlcTask Inputs/GVL_iXlinker.EtherCAT_Master_APSxxxx.Beckhoff_APS1xxx.A_0002_APS1003_5000_0016.FB_Inputs.F5_Y_Field <-> FB Inputs/F5 Y-Field
//     PlcTask Inputs/GVL_iXlinker.EtherCAT_Master_APSxxxx.Beckhoff_APS1xxx.A_0002_APS1003_5000_0016.FB_Inputs.F7_Y_Field <-> FB Inputs/F7 Y-Field
//     PlcTask Inputs/GVL_iXlinker.EtherCAT_Master_APSxxxx.Beckhoff_APS1xxx.A_0002_APS1003_5000_0016.FB_Inputs.F9_Y_Field <-> FB Inputs/F9 Y-Field
//     PlcTask Inputs/GVL_iXlinker.EtherCAT_Master_APSxxxx.Beckhoff_APS1xxx.A_0002_APS1003_5000_0016.FB_Inputs.F1_Z_Field <-> FB Inputs/F1 Z-Field
//     PlcTask Inputs/GVL_iXlinker.EtherCAT_Master_APSxxxx.Beckhoff_APS1xxx.A_0002_APS1003_5000_0016.FB_Inputs.F3_Z_Field <-> FB Inputs/F3 Z-Field
//     PlcTask Inputs/GVL_iXlinker.EtherCAT_Master_APSxxxx.Beckhoff_APS1xxx.A_0002_APS1003_5000_0016.FB_Inputs.F5_Z_Field <-> FB Inputs/F5 Z-Field
//     PlcTask Inputs/GVL_iXlinker.EtherCAT_Master_APSxxxx.Beckhoff_APS1xxx.A_0002_APS1003_5000_0016.FB_Inputs.F7_Z_Field <-> FB Inputs/F7 Z-Field
//     PlcTask Inputs/GVL_iXlinker.EtherCAT_Master_APSxxxx.Beckhoff_APS1xxx.A_0002_APS1003_5000_0016.FB_Inputs.F9_Z_Field <-> FB Inputs/F9 Z-Field
//     PlcTask Inputs/GVL_iXlinker.EtherCAT_Master_APSxxxx.Beckhoff_APS1xxx.A_0002_APS1003_5000_0016.FB_Inputs.G0_X_Field <-> FB Inputs/G0 X-Field
//     PlcTask Inputs/GVL_iXlinker.EtherCAT_Master_APSxxxx.Beckhoff_APS1xxx.A_0002_APS1003_5000_0016.FB_Inputs.G2_X_Field <-> FB Inputs/G2 X-Field
//     PlcTask Inputs/GVL_iXlinker.EtherCAT_Master_APSxxxx.Beckhoff_APS1xxx.A_0002_APS1003_5000_0016.FB_Inputs.G4_X_Field <-> FB Inputs/G4 X-Field
//     PlcTask Inputs/GVL_iXlinker.EtherCAT_Master_APSxxxx.Beckhoff_APS1xxx.A_0002_APS1003_5000_0016.FB_Inputs.G6_X_Field <-> FB Inputs/G6 X-Field
//     PlcTask Inputs/GVL_iXlinker.EtherCAT_Master_APSxxxx.Beckhoff_APS1xxx.A_0002_APS1003_5000_0016.FB_Inputs.G8_X_Field <-> FB Inputs/G8 X-Field
//     PlcTask Inputs/GVL_iXlinker.EtherCAT_Master_APSxxxx.Beckhoff_APS1xxx.A_0002_APS1003_5000_0016.FB_Inputs.G0_Y_Field <-> FB Inputs/G0 Y-Field
//     PlcTask Inputs/GVL_iXlinker.EtherCAT_Master_APSxxxx.Beckhoff_APS1xxx.A_0002_APS1003_5000_0016.FB_Inputs.G2_Y_Field <-> FB Inputs/G2 Y-Field
//     PlcTask Inputs/GVL_iXlinker.EtherCAT_Master_APSxxxx.Beckhoff_APS1xxx.A_0002_APS1003_5000_0016.FB_Inputs.G4_Y_Field <-> FB Inputs/G4 Y-Field
//     PlcTask Inputs/GVL_iXlinker.EtherCAT_Master_APSxxxx.Beckhoff_APS1xxx.A_0002_APS1003_5000_0016.FB_Inputs.G6_Y_Field <-> FB Inputs/G6 Y-Field
//     PlcTask Inputs/GVL_iXlinker.EtherCAT_Master_APSxxxx.Beckhoff_APS1xxx.A_0002_APS1003_5000_0016.FB_Inputs.G8_Y_Field <-> FB Inputs/G8 Y-Field
//     PlcTask Inputs/GVL_iXlinker.EtherCAT_Master_APSxxxx.Beckhoff_APS1xxx.A_0002_APS1003_5000_0016.FB_Inputs.G0_Z_Field <-> FB Inputs/G0 Z-Field
//     PlcTask Inputs/GVL_iXlinker.EtherCAT_Master_APSxxxx.Beckhoff_APS1xxx.A_0002_APS1003_5000_0016.FB_Inputs.G2_Z_Field <-> FB Inputs/G2 Z-Field
//     PlcTask Inputs/GVL_iXlinker.EtherCAT_Master_APSxxxx.Beckhoff_APS1xxx.A_0002_APS1003_5000_0016.FB_Inputs.G4_Z_Field <-> FB Inputs/G4 Z-Field
//     PlcTask Inputs/GVL_iXlinker.EtherCAT_Master_APSxxxx.Beckhoff_APS1xxx.A_0002_APS1003_5000_0016.FB_Inputs.G6_Z_Field <-> FB Inputs/G6 Z-Field
//     PlcTask Inputs/GVL_iXlinker.EtherCAT_Master_APSxxxx.Beckhoff_APS1xxx.A_0002_APS1003_5000_0016.FB_Inputs.G8_Z_Field <-> FB Inputs/G8 Z-Field
//     PlcTask Inputs/GVL_iXlinker.EtherCAT_Master_APSxxxx.Beckhoff_APS1xxx.A_0002_APS1003_5000_0016.FB_Inputs.H1_X_Field <-> FB Inputs/H1 X-Field
//     PlcTask Inputs/GVL_iXlinker.EtherCAT_Master_APSxxxx.Beckhoff_APS1xxx.A_0002_APS1003_5000_0016.FB_Inputs.H3_X_Field <-> FB Inputs/H3 X-Field
//     PlcTask Inputs/GVL_iXlinker.EtherCAT_Master_APSxxxx.Beckhoff_APS1xxx.A_0002_APS1003_5000_0016.FB_Inputs.H5_X_Field <-> FB Inputs/H5 X-Field
//     PlcTask Inputs/GVL_iXlinker.EtherCAT_Master_APSxxxx.Beckhoff_APS1xxx.A_0002_APS1003_5000_0016.FB_Inputs.H7_X_Field <-> FB Inputs/H7 X-Field
//     PlcTask Inputs/GVL_iXlinker.EtherCAT_Master_APSxxxx.Beckhoff_APS1xxx.A_0002_APS1003_5000_0016.FB_Inputs.H9_X_Field <-> FB Inputs/H9 X-Field
//     PlcTask Inputs/GVL_iXlinker.EtherCAT_Master_APSxxxx.Beckhoff_APS1xxx.A_0002_APS1003_5000_0016.FB_Inputs.H1_Y_Field <-> FB Inputs/H1 Y-Field
//     PlcTask Inputs/GVL_iXlinker.EtherCAT_Master_APSxxxx.Beckhoff_APS1xxx.A_0002_APS1003_5000_0016.FB_Inputs.H3_Y_Field <-> FB Inputs/H3 Y-Field
//     PlcTask Inputs/GVL_iXlinker.EtherCAT_Master_APSxxxx.Beckhoff_APS1xxx.A_0002_APS1003_5000_0016.FB_Inputs.H5_Y_Field <-> FB Inputs/H5 Y-Field
//     PlcTask Inputs/GVL_iXlinker.EtherCAT_Master_APSxxxx.Beckhoff_APS1xxx.A_0002_APS1003_5000_0016.FB_Inputs.H7_Y_Field <-> FB Inputs/H7 Y-Field
//     PlcTask Inputs/GVL_iXlinker.EtherCAT_Master_APSxxxx.Beckhoff_APS1xxx.A_0002_APS1003_5000_0016.FB_Inputs.H9_Y_Field <-> FB Inputs/H9 Y-Field
//     PlcTask Inputs/GVL_iXlinker.EtherCAT_Master_APSxxxx.Beckhoff_APS1xxx.A_0002_APS1003_5000_0016.FB_Inputs.H1_Z_Field <-> FB Inputs/H1 Z-Field
//     PlcTask Inputs/GVL_iXlinker.EtherCAT_Master_APSxxxx.Beckhoff_APS1xxx.A_0002_APS1003_5000_0016.FB_Inputs.H3_Z_Field <-> FB Inputs/H3 Z-Field
//     PlcTask Inputs/GVL_iXlinker.EtherCAT_Master_APSxxxx.Beckhoff_APS1xxx.A_0002_APS1003_5000_0016.FB_Inputs.H5_Z_Field <-> FB Inputs/H5 Z-Field
//     PlcTask Inputs/GVL_iXlinker.EtherCAT_Master_APSxxxx.Beckhoff_APS1xxx.A_0002_APS1003_5000_0016.FB_Inputs.H7_Z_Field <-> FB Inputs/H7 Z-Field
//     PlcTask Inputs/GVL_iXlinker.EtherCAT_Master_APSxxxx.Beckhoff_APS1xxx.A_0002_APS1003_5000_0016.FB_Inputs.H9_Z_Field <-> FB Inputs/H9 Z-Field
//     PlcTask Inputs/GVL_iXlinker.EtherCAT_Master_APSxxxx.Beckhoff_APS1xxx.A_0002_APS1003_5000_0016.FB_Inputs.I0_X_Field <-> FB Inputs/I0 X-Field
//     PlcTask Inputs/GVL_iXlinker.EtherCAT_Master_APSxxxx.Beckhoff_APS1xxx.A_0002_APS1003_5000_0016.FB_Inputs.I2_X_Field <-> FB Inputs/I2 X-Field
//     PlcTask Inputs/GVL_iXlinker.EtherCAT_Master_APSxxxx.Beckhoff_APS1xxx.A_0002_APS1003_5000_0016.FB_Inputs.I4_X_Field <-> FB Inputs/I4 X-Field
//     PlcTask Inputs/GVL_iXlinker.EtherCAT_Master_APSxxxx.Beckhoff_APS1xxx.A_0002_APS1003_5000_0016.FB_Inputs.I6_X_Field <-> FB Inputs/I6 X-Field
//     PlcTask Inputs/GVL_iXlinker.EtherCAT_Master_APSxxxx.Beckhoff_APS1xxx.A_0002_APS1003_5000_0016.FB_Inputs.I8_X_Field <-> FB Inputs/I8 X-Field
//     PlcTask Inputs/GVL_iXlinker.EtherCAT_Master_APSxxxx.Beckhoff_APS1xxx.A_0002_APS1003_5000_0016.FB_Inputs.I0_Y_Field <-> FB Inputs/I0 Y-Field
//     PlcTask Inputs/GVL_iXlinker.EtherCAT_Master_APSxxxx.Beckhoff_APS1xxx.A_0002_APS1003_5000_0016.FB_Inputs.I2_Y_Field <-> FB Inputs/I2 Y-Field
//     PlcTask Inputs/GVL_iXlinker.EtherCAT_Master_APSxxxx.Beckhoff_APS1xxx.A_0002_APS1003_5000_0016.FB_Inputs.I4_Y_Field <-> FB Inputs/I4 Y-Field
//     PlcTask Inputs/GVL_iXlinker.EtherCAT_Master_APSxxxx.Beckhoff_APS1xxx.A_0002_APS1003_5000_0016.FB_Inputs.I6_Y_Field <-> FB Inputs/I6 Y-Field
//     PlcTask Inputs/GVL_iXlinker.EtherCAT_Master_APSxxxx.Beckhoff_APS1xxx.A_0002_APS1003_5000_0016.FB_Inputs.I8_Y_Field <-> FB Inputs/I8 Y-Field
//     PlcTask Inputs/GVL_iXlinker.EtherCAT_Master_APSxxxx.Beckhoff_APS1xxx.A_0002_APS1003_5000_0016.FB_Inputs.I0_Z_Field <-> FB Inputs/I0 Z-Field
//     PlcTask Inputs/GVL_iXlinker.EtherCAT_Master_APSxxxx.Beckhoff_APS1xxx.A_0002_APS1003_5000_0016.FB_Inputs.I2_Z_Field <-> FB Inputs/I2 Z-Field
//     PlcTask Inputs/GVL_iXlinker.EtherCAT_Master_APSxxxx.Beckhoff_APS1xxx.A_0002_APS1003_5000_0016.FB_Inputs.I4_Z_Field <-> FB Inputs/I4 Z-Field
//     PlcTask Inputs/GVL_iXlinker.EtherCAT_Master_APSxxxx.Beckhoff_APS1xxx.A_0002_APS1003_5000_0016.FB_Inputs.I6_Z_Field <-> FB Inputs/I6 Z-Field
//     PlcTask Inputs/GVL_iXlinker.EtherCAT_Master_APSxxxx.Beckhoff_APS1xxx.A_0002_APS1003_5000_0016.FB_Inputs.I8_Z_Field <-> FB Inputs/I8 Z-Field
//     PlcTask Inputs/GVL_iXlinker.EtherCAT_Master_APSxxxx.Beckhoff_APS1xxx.A_0002_APS1003_5000_0016.FB_Inputs.J1_X_Field <-> FB Inputs/J1 X-Field
//     PlcTask Inputs/GVL_iXlinker.EtherCAT_Master_APSxxxx.Beckhoff_APS1xxx.A_0002_APS1003_5000_0016.FB_Inputs.J3_X_Field <-> FB Inputs/J3 X-Field
//     PlcTask Inputs/GVL_iXlinker.EtherCAT_Master_APSxxxx.Beckhoff_APS1xxx.A_0002_APS1003_5000_0016.FB_Inputs.J5_X_Field <-> FB Inputs/J5 X-Field
//     PlcTask Inputs/GVL_iXlinker.EtherCAT_Master_APSxxxx.Beckhoff_APS1xxx.A_0002_APS1003_5000_0016.FB_Inputs.J7_X_Field <-> FB Inputs/J7 X-Field
//     PlcTask Inputs/GVL_iXlinker.EtherCAT_Master_APSxxxx.Beckhoff_APS1xxx.A_0002_APS1003_5000_0016.FB_Inputs.J9_X_Field <-> FB Inputs/J9 X-Field
//     PlcTask Inputs/GVL_iXlinker.EtherCAT_Master_APSxxxx.Beckhoff_APS1xxx.A_0002_APS1003_5000_0016.FB_Inputs.J1_Y_Field <-> FB Inputs/J1 Y-Field
//     PlcTask Inputs/GVL_iXlinker.EtherCAT_Master_APSxxxx.Beckhoff_APS1xxx.A_0002_APS1003_5000_0016.FB_Inputs.J3_Y_Field <-> FB Inputs/J3 Y-Field
//     PlcTask Inputs/GVL_iXlinker.EtherCAT_Master_APSxxxx.Beckhoff_APS1xxx.A_0002_APS1003_5000_0016.FB_Inputs.J5_Y_Field <-> FB Inputs/J5 Y-Field
//     PlcTask Inputs/GVL_iXlinker.EtherCAT_Master_APSxxxx.Beckhoff_APS1xxx.A_0002_APS1003_5000_0016.FB_Inputs.J7_Y_Field <-> FB Inputs/J7 Y-Field
//     PlcTask Inputs/GVL_iXlinker.EtherCAT_Master_APSxxxx.Beckhoff_APS1xxx.A_0002_APS1003_5000_0016.FB_Inputs.J9_Y_Field <-> FB Inputs/J9 Y-Field
//     PlcTask Inputs/GVL_iXlinker.EtherCAT_Master_APSxxxx.Beckhoff_APS1xxx.A_0002_APS1003_5000_0016.FB_Inputs.J1_Z_Field <-> FB Inputs/J1 Z-Field
//     PlcTask Inputs/GVL_iXlinker.EtherCAT_Master_APSxxxx.Beckhoff_APS1xxx.A_0002_APS1003_5000_0016.FB_Inputs.J3_Z_Field <-> FB Inputs/J3 Z-Field
//     PlcTask Inputs/GVL_iXlinker.EtherCAT_Master_APSxxxx.Beckhoff_APS1xxx.A_0002_APS1003_5000_0016.FB_Inputs.J5_Z_Field <-> FB Inputs/J5 Z-Field
//     PlcTask Inputs/GVL_iXlinker.EtherCAT_Master_APSxxxx.Beckhoff_APS1xxx.A_0002_APS1003_5000_0016.FB_Inputs.J7_Z_Field <-> FB Inputs/J7 Z-Field
//     PlcTask Inputs/GVL_iXlinker.EtherCAT_Master_APSxxxx.Beckhoff_APS1xxx.A_0002_APS1003_5000_0016.FB_Inputs.J9_Z_Field <-> FB Inputs/J9 Z-Field
//     PlcTask Inputs/GVL_iXlinker.EtherCAT_Master_APSxxxx.Beckhoff_APS1xxx.A_0002_APS1003_5000_0016.WcState.WcState <-> WcState/WcState
//     PlcTask Inputs/GVL_iXlinker.EtherCAT_Master_APSxxxx.Beckhoff_APS1xxx.A_0002_APS1003_5000_0016.WcState.InputToggle <-> WcState/InputToggle
//     PlcTask Inputs/GVL_iXlinker.EtherCAT_Master_APSxxxx.Beckhoff_APS1xxx.A_0002_APS1003_5000_0016.InfoData.DcOutputShift <-> InfoData/DcOutputShift
//     PlcTask Inputs/GVL_iXlinker.EtherCAT_Master_APSxxxx.Beckhoff_APS1xxx.A_0002_APS1003_5000_0016.InfoData.DcInputShift <-> InfoData/DcInputShift
//     PlcTask Inputs/GVL_iXlinker.EtherCAT_Master_APSxxxx.Beckhoff_APS1xxx.A_0002_APS1003_5000_0016.InfoData.State <-> InfoData/State
//   PLC/PLC Instance <-> EtherCAT Master APSxxxx/Beckhoff APS4xxx
//     PlcTask Inputs/GVL_iXlinker.EtherCAT_Master_APSxxxx.Beckhoff_APS4xxx.InfoData.State <-> InfoData/State
//   PLC/PLC Instance <-> EtherCAT Master APSxxxx/Beckhoff APS4xxx/Beckhoff APS4xxxEK1122
//     PlcTask Inputs/GVL_iXlinker.EtherCAT_Master_APSxxxx.Beckhoff_APS4xxx.Beckhoff_APS4xxxEK1122.InfoData.State <-> InfoData/State
//   PLC/PLC Instance <-> EtherCAT Master APSxxxx/Beckhoff APS4xxx/Beckhoff APS4xxxEK1122/Beckhoff APS4xxxsub EK1100
//     PlcTask Inputs/GVL_iXlinker.EtherCAT_Master_APSxxxx.Beckhoff_APS4xxx.Beckhoff_APS4xxxEK1122.Beckhoff_APS4xxxsub_EK1100.InfoData.State <-> InfoData/State
//   PLC/PLC Instance <-> EtherCAT Master APSxxxx/Beckhoff APS4xxx/Beckhoff APS4xxxEK1122/A_0001(APS4322-7000-0017)
//     PlcTask Inputs/GVL_iXlinker.EtherCAT_Master_APSxxxx.Beckhoff_APS4xxx.Beckhoff_APS4xxxEK1122.A_0001_APS4322_7000_0017.APS_Inputs.StatusWord <-> APS Inputs/StatusWord
//     PlcTask Inputs/GVL_iXlinker.EtherCAT_Master_APSxxxx.Beckhoff_APS4xxx.Beckhoff_APS4xxxEK1122.A_0001_APS4322_7000_0017.APS_Inputs.Current_D_0X0 <-> APS Inputs/Current D 0X0
//     PlcTask Inputs/GVL_iXlinker.EtherCAT_Master_APSxxxx.Beckhoff_APS4xxx.Beckhoff_APS4xxxEK1122.A_0001_APS4322_7000_0017.APS_Inputs.Current_D_0X1 <-> APS Inputs/Current D 0X1
//     PlcTask Inputs/GVL_iXlinker.EtherCAT_Master_APSxxxx.Beckhoff_APS4xxx.Beckhoff_APS4xxxEK1122.A_0001_APS4322_7000_0017.APS_Inputs.Current_D_0X2 <-> APS Inputs/Current D 0X2
//     PlcTask Inputs/GVL_iXlinker.EtherCAT_Master_APSxxxx.Beckhoff_APS4xxx.Beckhoff_APS4xxxEK1122.A_0001_APS4322_7000_0017.APS_Inputs.Current_D_1X0 <-> APS Inputs/Current D 1X0
//     PlcTask Inputs/GVL_iXlinker.EtherCAT_Master_APSxxxx.Beckhoff_APS4xxx.Beckhoff_APS4xxxEK1122.A_0001_APS4322_7000_0017.APS_Inputs.Current_D_1X1 <-> APS Inputs/Current D 1X1
//     PlcTask Inputs/GVL_iXlinker.EtherCAT_Master_APSxxxx.Beckhoff_APS4xxx.Beckhoff_APS4xxxEK1122.A_0001_APS4322_7000_0017.APS_Inputs.Current_D_1X2 <-> APS Inputs/Current D 1X2
//     PlcTask Inputs/GVL_iXlinker.EtherCAT_Master_APSxxxx.Beckhoff_APS4xxx.Beckhoff_APS4xxxEK1122.A_0001_APS4322_7000_0017.APS_Inputs.Current_D_2X0 <-> APS Inputs/Current D 2X0
//     PlcTask Inputs/GVL_iXlinker.EtherCAT_Master_APSxxxx.Beckhoff_APS4xxx.Beckhoff_APS4xxxEK1122.A_0001_APS4322_7000_0017.APS_Inputs.Current_D_2X1 <-> APS Inputs/Current D 2X1
//     PlcTask Inputs/GVL_iXlinker.EtherCAT_Master_APSxxxx.Beckhoff_APS4xxx.Beckhoff_APS4xxxEK1122.A_0001_APS4322_7000_0017.APS_Inputs.Current_D_2X2 <-> APS Inputs/Current D 2X2
//     PlcTask Inputs/GVL_iXlinker.EtherCAT_Master_APSxxxx.Beckhoff_APS4xxx.Beckhoff_APS4xxxEK1122.A_0001_APS4322_7000_0017.APS_Inputs.Current_D_3X0 <-> APS Inputs/Current D 3X0
//     PlcTask Inputs/GVL_iXlinker.EtherCAT_Master_APSxxxx.Beckhoff_APS4xxx.Beckhoff_APS4xxxEK1122.A_0001_APS4322_7000_0017.APS_Inputs.Current_D_3X1 <-> APS Inputs/Current D 3X1
//     PlcTask Inputs/GVL_iXlinker.EtherCAT_Master_APSxxxx.Beckhoff_APS4xxx.Beckhoff_APS4xxxEK1122.A_0001_APS4322_7000_0017.APS_Inputs.Current_D_3X2 <-> APS Inputs/Current D 3X2
//     PlcTask Inputs/GVL_iXlinker.EtherCAT_Master_APSxxxx.Beckhoff_APS4xxx.Beckhoff_APS4xxxEK1122.A_0001_APS4322_7000_0017.APS_Inputs.Current_D_0Y0 <-> APS Inputs/Current D 0Y0
//     PlcTask Inputs/GVL_iXlinker.EtherCAT_Master_APSxxxx.Beckhoff_APS4xxx.Beckhoff_APS4xxxEK1122.A_0001_APS4322_7000_0017.APS_Inputs.Current_D_0Y1 <-> APS Inputs/Current D 0Y1
//     PlcTask Inputs/GVL_iXlinker.EtherCAT_Master_APSxxxx.Beckhoff_APS4xxx.Beckhoff_APS4xxxEK1122.A_0001_APS4322_7000_0017.APS_Inputs.Current_D_0Y2 <-> APS Inputs/Current D 0Y2
//     PlcTask Inputs/GVL_iXlinker.EtherCAT_Master_APSxxxx.Beckhoff_APS4xxx.Beckhoff_APS4xxxEK1122.A_0001_APS4322_7000_0017.APS_Inputs.Current_D_1Y0 <-> APS Inputs/Current D 1Y0
//     PlcTask Inputs/GVL_iXlinker.EtherCAT_Master_APSxxxx.Beckhoff_APS4xxx.Beckhoff_APS4xxxEK1122.A_0001_APS4322_7000_0017.APS_Inputs.Current_D_1Y1 <-> APS Inputs/Current D 1Y1
//     PlcTask Inputs/GVL_iXlinker.EtherCAT_Master_APSxxxx.Beckhoff_APS4xxx.Beckhoff_APS4xxxEK1122.A_0001_APS4322_7000_0017.APS_Inputs.Current_D_1Y2 <-> APS Inputs/Current D 1Y2
//     PlcTask Inputs/GVL_iXlinker.EtherCAT_Master_APSxxxx.Beckhoff_APS4xxx.Beckhoff_APS4xxxEK1122.A_0001_APS4322_7000_0017.APS_Inputs.Current_D_2Y0 <-> APS Inputs/Current D 2Y0
//     PlcTask Inputs/GVL_iXlinker.EtherCAT_Master_APSxxxx.Beckhoff_APS4xxx.Beckhoff_APS4xxxEK1122.A_0001_APS4322_7000_0017.APS_Inputs.Current_D_2Y1 <-> APS Inputs/Current D 2Y1
//     PlcTask Inputs/GVL_iXlinker.EtherCAT_Master_APSxxxx.Beckhoff_APS4xxx.Beckhoff_APS4xxxEK1122.A_0001_APS4322_7000_0017.APS_Inputs.Current_D_2Y2 <-> APS Inputs/Current D 2Y2
//     PlcTask Inputs/GVL_iXlinker.EtherCAT_Master_APSxxxx.Beckhoff_APS4xxx.Beckhoff_APS4xxxEK1122.A_0001_APS4322_7000_0017.APS_Inputs.Current_D_3Y0 <-> APS Inputs/Current D 3Y0
//     PlcTask Inputs/GVL_iXlinker.EtherCAT_Master_APSxxxx.Beckhoff_APS4xxx.Beckhoff_APS4xxxEK1122.A_0001_APS4322_7000_0017.APS_Inputs.Current_D_3Y1 <-> APS Inputs/Current D 3Y1
//     PlcTask Inputs/GVL_iXlinker.EtherCAT_Master_APSxxxx.Beckhoff_APS4xxx.Beckhoff_APS4xxxEK1122.A_0001_APS4322_7000_0017.APS_Inputs.Current_D_3Y2 <-> APS Inputs/Current D 3Y2
//     PlcTask Inputs/GVL_iXlinker.EtherCAT_Master_APSxxxx.Beckhoff_APS4xxx.Beckhoff_APS4xxxEK1122.A_0001_APS4322_7000_0017.APS_Inputs.Current_Q_0X0 <-> APS Inputs/Current Q 0X0
//     PlcTask Inputs/GVL_iXlinker.EtherCAT_Master_APSxxxx.Beckhoff_APS4xxx.Beckhoff_APS4xxxEK1122.A_0001_APS4322_7000_0017.APS_Inputs.Current_Q_0X1 <-> APS Inputs/Current Q 0X1
//     PlcTask Inputs/GVL_iXlinker.EtherCAT_Master_APSxxxx.Beckhoff_APS4xxx.Beckhoff_APS4xxxEK1122.A_0001_APS4322_7000_0017.APS_Inputs.Current_Q_0X2 <-> APS Inputs/Current Q 0X2
//     PlcTask Inputs/GVL_iXlinker.EtherCAT_Master_APSxxxx.Beckhoff_APS4xxx.Beckhoff_APS4xxxEK1122.A_0001_APS4322_7000_0017.APS_Inputs.Current_Q_1X0 <-> APS Inputs/Current Q 1X0
//     PlcTask Inputs/GVL_iXlinker.EtherCAT_Master_APSxxxx.Beckhoff_APS4xxx.Beckhoff_APS4xxxEK1122.A_0001_APS4322_7000_0017.APS_Inputs.Current_Q_1X1 <-> APS Inputs/Current Q 1X1
//     PlcTask Inputs/GVL_iXlinker.EtherCAT_Master_APSxxxx.Beckhoff_APS4xxx.Beckhoff_APS4xxxEK1122.A_0001_APS4322_7000_0017.APS_Inputs.Current_Q_1X2 <-> APS Inputs/Current Q 1X2
//     PlcTask Inputs/GVL_iXlinker.EtherCAT_Master_APSxxxx.Beckhoff_APS4xxx.Beckhoff_APS4xxxEK1122.A_0001_APS4322_7000_0017.APS_Inputs.Current_Q_2X0 <-> APS Inputs/Current Q 2X0
//     PlcTask Inputs/GVL_iXlinker.EtherCAT_Master_APSxxxx.Beckhoff_APS4xxx.Beckhoff_APS4xxxEK1122.A_0001_APS4322_7000_0017.APS_Inputs.Current_Q_2X1 <-> APS Inputs/Current Q 2X1
//     PlcTask Inputs/GVL_iXlinker.EtherCAT_Master_APSxxxx.Beckhoff_APS4xxx.Beckhoff_APS4xxxEK1122.A_0001_APS4322_7000_0017.APS_Inputs.Current_Q_2X2 <-> APS Inputs/Current Q 2X2
//     PlcTask Inputs/GVL_iXlinker.EtherCAT_Master_APSxxxx.Beckhoff_APS4xxx.Beckhoff_APS4xxxEK1122.A_0001_APS4322_7000_0017.APS_Inputs.Current_Q_3X0 <-> APS Inputs/Current Q 3X0
//     PlcTask Inputs/GVL_iXlinker.EtherCAT_Master_APSxxxx.Beckhoff_APS4xxx.Beckhoff_APS4xxxEK1122.A_0001_APS4322_7000_0017.APS_Inputs.Current_Q_3X1 <-> APS Inputs/Current Q 3X1
//     PlcTask Inputs/GVL_iXlinker.EtherCAT_Master_APSxxxx.Beckhoff_APS4xxx.Beckhoff_APS4xxxEK1122.A_0001_APS4322_7000_0017.APS_Inputs.Current_Q_3X2 <-> APS Inputs/Current Q 3X2
//     PlcTask Inputs/GVL_iXlinker.EtherCAT_Master_APSxxxx.Beckhoff_APS4xxx.Beckhoff_APS4xxxEK1122.A_0001_APS4322_7000_0017.APS_Inputs.Current_Q_0Y0 <-> APS Inputs/Current Q 0Y0
//     PlcTask Inputs/GVL_iXlinker.EtherCAT_Master_APSxxxx.Beckhoff_APS4xxx.Beckhoff_APS4xxxEK1122.A_0001_APS4322_7000_0017.APS_Inputs.Current_Q_0Y1 <-> APS Inputs/Current Q 0Y1
//     PlcTask Inputs/GVL_iXlinker.EtherCAT_Master_APSxxxx.Beckhoff_APS4xxx.Beckhoff_APS4xxxEK1122.A_0001_APS4322_7000_0017.APS_Inputs.Current_Q_0Y2 <-> APS Inputs/Current Q 0Y2
//     PlcTask Inputs/GVL_iXlinker.EtherCAT_Master_APSxxxx.Beckhoff_APS4xxx.Beckhoff_APS4xxxEK1122.A_0001_APS4322_7000_0017.APS_Inputs.Current_Q_1Y0 <-> APS Inputs/Current Q 1Y0
//     PlcTask Inputs/GVL_iXlinker.EtherCAT_Master_APSxxxx.Beckhoff_APS4xxx.Beckhoff_APS4xxxEK1122.A_0001_APS4322_7000_0017.APS_Inputs.Current_Q_1Y1 <-> APS Inputs/Current Q 1Y1
//     PlcTask Inputs/GVL_iXlinker.EtherCAT_Master_APSxxxx.Beckhoff_APS4xxx.Beckhoff_APS4xxxEK1122.A_0001_APS4322_7000_0017.APS_Inputs.Current_Q_1Y2 <-> APS Inputs/Current Q 1Y2
//     PlcTask Inputs/GVL_iXlinker.EtherCAT_Master_APSxxxx.Beckhoff_APS4xxx.Beckhoff_APS4xxxEK1122.A_0001_APS4322_7000_0017.APS_Inputs.Current_Q_2Y0 <-> APS Inputs/Current Q 2Y0
//     PlcTask Inputs/GVL_iXlinker.EtherCAT_Master_APSxxxx.Beckhoff_APS4xxx.Beckhoff_APS4xxxEK1122.A_0001_APS4322_7000_0017.APS_Inputs.Current_Q_2Y1 <-> APS Inputs/Current Q 2Y1
//     PlcTask Inputs/GVL_iXlinker.EtherCAT_Master_APSxxxx.Beckhoff_APS4xxx.Beckhoff_APS4xxxEK1122.A_0001_APS4322_7000_0017.APS_Inputs.Current_Q_2Y2 <-> APS Inputs/Current Q 2Y2
//     PlcTask Inputs/GVL_iXlinker.EtherCAT_Master_APSxxxx.Beckhoff_APS4xxx.Beckhoff_APS4xxxEK1122.A_0001_APS4322_7000_0017.APS_Inputs.Current_Q_3Y0 <-> APS Inputs/Current Q 3Y0
//     PlcTask Inputs/GVL_iXlinker.EtherCAT_Master_APSxxxx.Beckhoff_APS4xxx.Beckhoff_APS4xxxEK1122.A_0001_APS4322_7000_0017.APS_Inputs.Current_Q_3Y1 <-> APS Inputs/Current Q 3Y1
//     PlcTask Inputs/GVL_iXlinker.EtherCAT_Master_APSxxxx.Beckhoff_APS4xxx.Beckhoff_APS4xxxEK1122.A_0001_APS4322_7000_0017.APS_Inputs.Current_Q_3Y2 <-> APS Inputs/Current Q 3Y2
//     PlcTask Inputs/GVL_iXlinker.EtherCAT_Master_APSxxxx.Beckhoff_APS4xxx.Beckhoff_APS4xxxEK1122.A_0001_APS4322_7000_0017.APS_Diagdata.DC_Link_Voltage <-> APS Diagdata/DC Link Voltage
//     PlcTask Inputs/GVL_iXlinker.EtherCAT_Master_APSxxxx.Beckhoff_APS4xxx.Beckhoff_APS4xxxEK1122.A_0001_APS4322_7000_0017.APS_Diagdata.Power_supply_current <-> APS Diagdata/Power supply current
//     PlcTask Inputs/GVL_iXlinker.EtherCAT_Master_APSxxxx.Beckhoff_APS4xxx.Beckhoff_APS4xxxEK1122.A_0001_APS4322_7000_0017.APS_Comm_Inputs.CommStatusWord <-> APS Comm Inputs/CommStatusWord
//     PlcTask Inputs/GVL_iXlinker.EtherCAT_Master_APSxxxx.Beckhoff_APS4xxx.Beckhoff_APS4xxxEK1122.A_0001_APS4322_7000_0017.APS_Comm_Inputs.Data[0] <-> APS Comm Inputs/Data 1
//     PlcTask Inputs/GVL_iXlinker.EtherCAT_Master_APSxxxx.Beckhoff_APS4xxx.Beckhoff_APS4xxxEK1122.A_0001_APS4322_7000_0017.APS_Comm_Inputs.Data[1] <-> APS Comm Inputs/Data 2
//     PlcTask Inputs/GVL_iXlinker.EtherCAT_Master_APSxxxx.Beckhoff_APS4xxx.Beckhoff_APS4xxxEK1122.A_0001_APS4322_7000_0017.APS_Comm_Inputs.Data[2] <-> APS Comm Inputs/Data 3
//     PlcTask Inputs/GVL_iXlinker.EtherCAT_Master_APSxxxx.Beckhoff_APS4xxx.Beckhoff_APS4xxxEK1122.A_0001_APS4322_7000_0017.APS_Comm_Inputs.Data[3] <-> APS Comm Inputs/Data 4
//     PlcTask Outputs/GVL_iXlinker.EtherCAT_Master_APSxxxx.Beckhoff_APS4xxx.Beckhoff_APS4xxxEK1122.A_0001_APS4322_7000_0017.APS_Outputs.ControlWord <-> APS Outputs/ControlWord
//     PlcTask Outputs/GVL_iXlinker.EtherCAT_Master_APSxxxx.Beckhoff_APS4xxx.Beckhoff_APS4xxxEK1122.A_0001_APS4322_7000_0017.APS_Outputs.Current_D_0X0 <-> APS Outputs/Current D 0X0
//     PlcTask Outputs/GVL_iXlinker.EtherCAT_Master_APSxxxx.Beckhoff_APS4xxx.Beckhoff_APS4xxxEK1122.A_0001_APS4322_7000_0017.APS_Outputs.Current_D_0X1 <-> APS Outputs/Current D 0X1
//     PlcTask Outputs/GVL_iXlinker.EtherCAT_Master_APSxxxx.Beckhoff_APS4xxx.Beckhoff_APS4xxxEK1122.A_0001_APS4322_7000_0017.APS_Outputs.Current_D_0X2 <-> APS Outputs/Current D 0X2
//     PlcTask Outputs/GVL_iXlinker.EtherCAT_Master_APSxxxx.Beckhoff_APS4xxx.Beckhoff_APS4xxxEK1122.A_0001_APS4322_7000_0017.APS_Outputs.Current_D_1X0 <-> APS Outputs/Current D 1X0
//     PlcTask Outputs/GVL_iXlinker.EtherCAT_Master_APSxxxx.Beckhoff_APS4xxx.Beckhoff_APS4xxxEK1122.A_0001_APS4322_7000_0017.APS_Outputs.Current_D_1X1 <-> APS Outputs/Current D 1X1
//     PlcTask Outputs/GVL_iXlinker.EtherCAT_Master_APSxxxx.Beckhoff_APS4xxx.Beckhoff_APS4xxxEK1122.A_0001_APS4322_7000_0017.APS_Outputs.Current_D_1X2 <-> APS Outputs/Current D 1X2
//     PlcTask Outputs/GVL_iXlinker.EtherCAT_Master_APSxxxx.Beckhoff_APS4xxx.Beckhoff_APS4xxxEK1122.A_0001_APS4322_7000_0017.APS_Outputs.Current_D_2X0 <-> APS Outputs/Current D 2X0
//     PlcTask Outputs/GVL_iXlinker.EtherCAT_Master_APSxxxx.Beckhoff_APS4xxx.Beckhoff_APS4xxxEK1122.A_0001_APS4322_7000_0017.APS_Outputs.Current_D_2X1 <-> APS Outputs/Current D 2X1
//     PlcTask Outputs/GVL_iXlinker.EtherCAT_Master_APSxxxx.Beckhoff_APS4xxx.Beckhoff_APS4xxxEK1122.A_0001_APS4322_7000_0017.APS_Outputs.Current_D_2X2 <-> APS Outputs/Current D 2X2
//     PlcTask Outputs/GVL_iXlinker.EtherCAT_Master_APSxxxx.Beckhoff_APS4xxx.Beckhoff_APS4xxxEK1122.A_0001_APS4322_7000_0017.APS_Outputs.Current_D_3X0 <-> APS Outputs/Current D 3X0
//     PlcTask Outputs/GVL_iXlinker.EtherCAT_Master_APSxxxx.Beckhoff_APS4xxx.Beckhoff_APS4xxxEK1122.A_0001_APS4322_7000_0017.APS_Outputs.Current_D_3X1 <-> APS Outputs/Current D 3X1
//     PlcTask Outputs/GVL_iXlinker.EtherCAT_Master_APSxxxx.Beckhoff_APS4xxx.Beckhoff_APS4xxxEK1122.A_0001_APS4322_7000_0017.APS_Outputs.Current_D_3X2 <-> APS Outputs/Current D 3X2
//     PlcTask Outputs/GVL_iXlinker.EtherCAT_Master_APSxxxx.Beckhoff_APS4xxx.Beckhoff_APS4xxxEK1122.A_0001_APS4322_7000_0017.APS_Outputs.Current_D_0Y0 <-> APS Outputs/Current D 0Y0
//     PlcTask Outputs/GVL_iXlinker.EtherCAT_Master_APSxxxx.Beckhoff_APS4xxx.Beckhoff_APS4xxxEK1122.A_0001_APS4322_7000_0017.APS_Outputs.Current_D_0Y1 <-> APS Outputs/Current D 0Y1
//     PlcTask Outputs/GVL_iXlinker.EtherCAT_Master_APSxxxx.Beckhoff_APS4xxx.Beckhoff_APS4xxxEK1122.A_0001_APS4322_7000_0017.APS_Outputs.Current_D_0Y2 <-> APS Outputs/Current D 0Y2
//     PlcTask Outputs/GVL_iXlinker.EtherCAT_Master_APSxxxx.Beckhoff_APS4xxx.Beckhoff_APS4xxxEK1122.A_0001_APS4322_7000_0017.APS_Outputs.Current_D_1Y0 <-> APS Outputs/Current D 1Y0
//     PlcTask Outputs/GVL_iXlinker.EtherCAT_Master_APSxxxx.Beckhoff_APS4xxx.Beckhoff_APS4xxxEK1122.A_0001_APS4322_7000_0017.APS_Outputs.Current_D_1Y1 <-> APS Outputs/Current D 1Y1
//     PlcTask Outputs/GVL_iXlinker.EtherCAT_Master_APSxxxx.Beckhoff_APS4xxx.Beckhoff_APS4xxxEK1122.A_0001_APS4322_7000_0017.APS_Outputs.Current_D_1Y2 <-> APS Outputs/Current D 1Y2
//     PlcTask Outputs/GVL_iXlinker.EtherCAT_Master_APSxxxx.Beckhoff_APS4xxx.Beckhoff_APS4xxxEK1122.A_0001_APS4322_7000_0017.APS_Outputs.Current_D_2Y0 <-> APS Outputs/Current D 2Y0
//     PlcTask Outputs/GVL_iXlinker.EtherCAT_Master_APSxxxx.Beckhoff_APS4xxx.Beckhoff_APS4xxxEK1122.A_0001_APS4322_7000_0017.APS_Outputs.Current_D_2Y1 <-> APS Outputs/Current D 2Y1
//     PlcTask Outputs/GVL_iXlinker.EtherCAT_Master_APSxxxx.Beckhoff_APS4xxx.Beckhoff_APS4xxxEK1122.A_0001_APS4322_7000_0017.APS_Outputs.Current_D_2Y2 <-> APS Outputs/Current D 2Y2
//     PlcTask Outputs/GVL_iXlinker.EtherCAT_Master_APSxxxx.Beckhoff_APS4xxx.Beckhoff_APS4xxxEK1122.A_0001_APS4322_7000_0017.APS_Outputs.Current_D_3Y0 <-> APS Outputs/Current D 3Y0
//     PlcTask Outputs/GVL_iXlinker.EtherCAT_Master_APSxxxx.Beckhoff_APS4xxx.Beckhoff_APS4xxxEK1122.A_0001_APS4322_7000_0017.APS_Outputs.Current_D_3Y1 <-> APS Outputs/Current D 3Y1
//     PlcTask Outputs/GVL_iXlinker.EtherCAT_Master_APSxxxx.Beckhoff_APS4xxx.Beckhoff_APS4xxxEK1122.A_0001_APS4322_7000_0017.APS_Outputs.Current_D_3Y2 <-> APS Outputs/Current D 3Y2
//     PlcTask Outputs/GVL_iXlinker.EtherCAT_Master_APSxxxx.Beckhoff_APS4xxx.Beckhoff_APS4xxxEK1122.A_0001_APS4322_7000_0017.APS_Outputs.Current_Q_0X0 <-> APS Outputs/Current Q 0X0
//     PlcTask Outputs/GVL_iXlinker.EtherCAT_Master_APSxxxx.Beckhoff_APS4xxx.Beckhoff_APS4xxxEK1122.A_0001_APS4322_7000_0017.APS_Outputs.Current_Q_0X1 <-> APS Outputs/Current Q 0X1
//     PlcTask Outputs/GVL_iXlinker.EtherCAT_Master_APSxxxx.Beckhoff_APS4xxx.Beckhoff_APS4xxxEK1122.A_0001_APS4322_7000_0017.APS_Outputs.Current_Q_0X2 <-> APS Outputs/Current Q 0X2
//     PlcTask Outputs/GVL_iXlinker.EtherCAT_Master_APSxxxx.Beckhoff_APS4xxx.Beckhoff_APS4xxxEK1122.A_0001_APS4322_7000_0017.APS_Outputs.Current_Q_1X0 <-> APS Outputs/Current Q 1X0
//     PlcTask Outputs/GVL_iXlinker.EtherCAT_Master_APSxxxx.Beckhoff_APS4xxx.Beckhoff_APS4xxxEK1122.A_0001_APS4322_7000_0017.APS_Outputs.Current_Q_1X1 <-> APS Outputs/Current Q 1X1
//     PlcTask Outputs/GVL_iXlinker.EtherCAT_Master_APSxxxx.Beckhoff_APS4xxx.Beckhoff_APS4xxxEK1122.A_0001_APS4322_7000_0017.APS_Outputs.Current_Q_1X2 <-> APS Outputs/Current Q 1X2
//     PlcTask Outputs/GVL_iXlinker.EtherCAT_Master_APSxxxx.Beckhoff_APS4xxx.Beckhoff_APS4xxxEK1122.A_0001_APS4322_7000_0017.APS_Outputs.Current_Q_2X0 <-> APS Outputs/Current Q 2X0
//     PlcTask Outputs/GVL_iXlinker.EtherCAT_Master_APSxxxx.Beckhoff_APS4xxx.Beckhoff_APS4xxxEK1122.A_0001_APS4322_7000_0017.APS_Outputs.Current_Q_2X1 <-> APS Outputs/Current Q 2X1
//     PlcTask Outputs/GVL_iXlinker.EtherCAT_Master_APSxxxx.Beckhoff_APS4xxx.Beckhoff_APS4xxxEK1122.A_0001_APS4322_7000_0017.APS_Outputs.Current_Q_2X2 <-> APS Outputs/Current Q 2X2
//     PlcTask Outputs/GVL_iXlinker.EtherCAT_Master_APSxxxx.Beckhoff_APS4xxx.Beckhoff_APS4xxxEK1122.A_0001_APS4322_7000_0017.APS_Outputs.Current_Q_3X0 <-> APS Outputs/Current Q 3X0
//     PlcTask Outputs/GVL_iXlinker.EtherCAT_Master_APSxxxx.Beckhoff_APS4xxx.Beckhoff_APS4xxxEK1122.A_0001_APS4322_7000_0017.APS_Outputs.Current_Q_3X1 <-> APS Outputs/Current Q 3X1
//     PlcTask Outputs/GVL_iXlinker.EtherCAT_Master_APSxxxx.Beckhoff_APS4xxx.Beckhoff_APS4xxxEK1122.A_0001_APS4322_7000_0017.APS_Outputs.Current_Q_3X2 <-> APS Outputs/Current Q 3X2
//     PlcTask Outputs/GVL_iXlinker.EtherCAT_Master_APSxxxx.Beckhoff_APS4xxx.Beckhoff_APS4xxxEK1122.A_0001_APS4322_7000_0017.APS_Outputs.Current_Q_0Y0 <-> APS Outputs/Current Q 0Y0
//     PlcTask Outputs/GVL_iXlinker.EtherCAT_Master_APSxxxx.Beckhoff_APS4xxx.Beckhoff_APS4xxxEK1122.A_0001_APS4322_7000_0017.APS_Outputs.Current_Q_0Y1 <-> APS Outputs/Current Q 0Y1
//     PlcTask Outputs/GVL_iXlinker.EtherCAT_Master_APSxxxx.Beckhoff_APS4xxx.Beckhoff_APS4xxxEK1122.A_0001_APS4322_7000_0017.APS_Outputs.Current_Q_0Y2 <-> APS Outputs/Current Q 0Y2
//     PlcTask Outputs/GVL_iXlinker.EtherCAT_Master_APSxxxx.Beckhoff_APS4xxx.Beckhoff_APS4xxxEK1122.A_0001_APS4322_7000_0017.APS_Outputs.Current_Q_1Y0 <-> APS Outputs/Current Q 1Y0
//     PlcTask Outputs/GVL_iXlinker.EtherCAT_Master_APSxxxx.Beckhoff_APS4xxx.Beckhoff_APS4xxxEK1122.A_0001_APS4322_7000_0017.APS_Outputs.Current_Q_1Y1 <-> APS Outputs/Current Q 1Y1
//     PlcTask Outputs/GVL_iXlinker.EtherCAT_Master_APSxxxx.Beckhoff_APS4xxx.Beckhoff_APS4xxxEK1122.A_0001_APS4322_7000_0017.APS_Outputs.Current_Q_1Y2 <-> APS Outputs/Current Q 1Y2
//     PlcTask Outputs/GVL_iXlinker.EtherCAT_Master_APSxxxx.Beckhoff_APS4xxx.Beckhoff_APS4xxxEK1122.A_0001_APS4322_7000_0017.APS_Outputs.Current_Q_2Y0 <-> APS Outputs/Current Q 2Y0
//     PlcTask Outputs/GVL_iXlinker.EtherCAT_Master_APSxxxx.Beckhoff_APS4xxx.Beckhoff_APS4xxxEK1122.A_0001_APS4322_7000_0017.APS_Outputs.Current_Q_2Y1 <-> APS Outputs/Current Q 2Y1
//     PlcTask Outputs/GVL_iXlinker.EtherCAT_Master_APSxxxx.Beckhoff_APS4xxx.Beckhoff_APS4xxxEK1122.A_0001_APS4322_7000_0017.APS_Outputs.Current_Q_2Y2 <-> APS Outputs/Current Q 2Y2
//     PlcTask Outputs/GVL_iXlinker.EtherCAT_Master_APSxxxx.Beckhoff_APS4xxx.Beckhoff_APS4xxxEK1122.A_0001_APS4322_7000_0017.APS_Outputs.Current_Q_3Y0 <-> APS Outputs/Current Q 3Y0
//     PlcTask Outputs/GVL_iXlinker.EtherCAT_Master_APSxxxx.Beckhoff_APS4xxx.Beckhoff_APS4xxxEK1122.A_0001_APS4322_7000_0017.APS_Outputs.Current_Q_3Y1 <-> APS Outputs/Current Q 3Y1
//     PlcTask Outputs/GVL_iXlinker.EtherCAT_Master_APSxxxx.Beckhoff_APS4xxx.Beckhoff_APS4xxxEK1122.A_0001_APS4322_7000_0017.APS_Outputs.Current_Q_3Y2 <-> APS Outputs/Current Q 3Y2
//     PlcTask Outputs/GVL_iXlinker.EtherCAT_Master_APSxxxx.Beckhoff_APS4xxx.Beckhoff_APS4xxxEK1122.A_0001_APS4322_7000_0017.APS_Outputs.PhiE_0X0 <-> APS Outputs/PhiE 0X0
//     PlcTask Outputs/GVL_iXlinker.EtherCAT_Master_APSxxxx.Beckhoff_APS4xxx.Beckhoff_APS4xxxEK1122.A_0001_APS4322_7000_0017.APS_Outputs.PhiE_0X1 <-> APS Outputs/PhiE 0X1
//     PlcTask Outputs/GVL_iXlinker.EtherCAT_Master_APSxxxx.Beckhoff_APS4xxx.Beckhoff_APS4xxxEK1122.A_0001_APS4322_7000_0017.APS_Outputs.PhiE_0X2 <-> APS Outputs/PhiE 0X2
//     PlcTask Outputs/GVL_iXlinker.EtherCAT_Master_APSxxxx.Beckhoff_APS4xxx.Beckhoff_APS4xxxEK1122.A_0001_APS4322_7000_0017.APS_Outputs.PhiE_1X0 <-> APS Outputs/PhiE 1X0
//     PlcTask Outputs/GVL_iXlinker.EtherCAT_Master_APSxxxx.Beckhoff_APS4xxx.Beckhoff_APS4xxxEK1122.A_0001_APS4322_7000_0017.APS_Outputs.PhiE_1X1 <-> APS Outputs/PhiE 1X1
//     PlcTask Outputs/GVL_iXlinker.EtherCAT_Master_APSxxxx.Beckhoff_APS4xxx.Beckhoff_APS4xxxEK1122.A_0001_APS4322_7000_0017.APS_Outputs.PhiE_1X2 <-> APS Outputs/PhiE 1X2
//     PlcTask Outputs/GVL_iXlinker.EtherCAT_Master_APSxxxx.Beckhoff_APS4xxx.Beckhoff_APS4xxxEK1122.A_0001_APS4322_7000_0017.APS_Outputs.PhiE_2X0 <-> APS Outputs/PhiE 2X0
//     PlcTask Outputs/GVL_iXlinker.EtherCAT_Master_APSxxxx.Beckhoff_APS4xxx.Beckhoff_APS4xxxEK1122.A_0001_APS4322_7000_0017.APS_Outputs.PhiE_2X1 <-> APS Outputs/PhiE 2X1
//     PlcTask Outputs/GVL_iXlinker.EtherCAT_Master_APSxxxx.Beckhoff_APS4xxx.Beckhoff_APS4xxxEK1122.A_0001_APS4322_7000_0017.APS_Outputs.PhiE_2X2 <-> APS Outputs/PhiE 2X2
//     PlcTask Outputs/GVL_iXlinker.EtherCAT_Master_APSxxxx.Beckhoff_APS4xxx.Beckhoff_APS4xxxEK1122.A_0001_APS4322_7000_0017.APS_Outputs.PhiE_3X0 <-> APS Outputs/PhiE 3X0
//     PlcTask Outputs/GVL_iXlinker.EtherCAT_Master_APSxxxx.Beckhoff_APS4xxx.Beckhoff_APS4xxxEK1122.A_0001_APS4322_7000_0017.APS_Outputs.PhiE_3X1 <-> APS Outputs/PhiE 3X1
//     PlcTask Outputs/GVL_iXlinker.EtherCAT_Master_APSxxxx.Beckhoff_APS4xxx.Beckhoff_APS4xxxEK1122.A_0001_APS4322_7000_0017.APS_Outputs.PhiE_3X2 <-> APS Outputs/PhiE 3X2
//     PlcTask Outputs/GVL_iXlinker.EtherCAT_Master_APSxxxx.Beckhoff_APS4xxx.Beckhoff_APS4xxxEK1122.A_0001_APS4322_7000_0017.APS_Outputs.PhiE_0Y0 <-> APS Outputs/PhiE 0Y0
//     PlcTask Outputs/GVL_iXlinker.EtherCAT_Master_APSxxxx.Beckhoff_APS4xxx.Beckhoff_APS4xxxEK1122.A_0001_APS4322_7000_0017.APS_Outputs.PhiE_0Y1 <-> APS Outputs/PhiE 0Y1
//     PlcTask Outputs/GVL_iXlinker.EtherCAT_Master_APSxxxx.Beckhoff_APS4xxx.Beckhoff_APS4xxxEK1122.A_0001_APS4322_7000_0017.APS_Outputs.PhiE_0Y2 <-> APS Outputs/PhiE 0Y2
//     PlcTask Outputs/GVL_iXlinker.EtherCAT_Master_APSxxxx.Beckhoff_APS4xxx.Beckhoff_APS4xxxEK1122.A_0001_APS4322_7000_0017.APS_Outputs.PhiE_1Y0 <-> APS Outputs/PhiE 1Y0
//     PlcTask Outputs/GVL_iXlinker.EtherCAT_Master_APSxxxx.Beckhoff_APS4xxx.Beckhoff_APS4xxxEK1122.A_0001_APS4322_7000_0017.APS_Outputs.PhiE_1Y1 <-> APS Outputs/PhiE 1Y1
//     PlcTask Outputs/GVL_iXlinker.EtherCAT_Master_APSxxxx.Beckhoff_APS4xxx.Beckhoff_APS4xxxEK1122.A_0001_APS4322_7000_0017.APS_Outputs.PhiE_1Y2 <-> APS Outputs/PhiE 1Y2
//     PlcTask Outputs/GVL_iXlinker.EtherCAT_Master_APSxxxx.Beckhoff_APS4xxx.Beckhoff_APS4xxxEK1122.A_0001_APS4322_7000_0017.APS_Outputs.PhiE_2Y0 <-> APS Outputs/PhiE 2Y0
//     PlcTask Outputs/GVL_iXlinker.EtherCAT_Master_APSxxxx.Beckhoff_APS4xxx.Beckhoff_APS4xxxEK1122.A_0001_APS4322_7000_0017.APS_Outputs.PhiE_2Y1 <-> APS Outputs/PhiE 2Y1
//     PlcTask Outputs/GVL_iXlinker.EtherCAT_Master_APSxxxx.Beckhoff_APS4xxx.Beckhoff_APS4xxxEK1122.A_0001_APS4322_7000_0017.APS_Outputs.PhiE_2Y2 <-> APS Outputs/PhiE 2Y2
//     PlcTask Outputs/GVL_iXlinker.EtherCAT_Master_APSxxxx.Beckhoff_APS4xxx.Beckhoff_APS4xxxEK1122.A_0001_APS4322_7000_0017.APS_Outputs.PhiE_3Y0 <-> APS Outputs/PhiE 3Y0
//     PlcTask Outputs/GVL_iXlinker.EtherCAT_Master_APSxxxx.Beckhoff_APS4xxx.Beckhoff_APS4xxxEK1122.A_0001_APS4322_7000_0017.APS_Outputs.PhiE_3Y1 <-> APS Outputs/PhiE 3Y1
//     PlcTask Outputs/GVL_iXlinker.EtherCAT_Master_APSxxxx.Beckhoff_APS4xxx.Beckhoff_APS4xxxEK1122.A_0001_APS4322_7000_0017.APS_Outputs.PhiE_3Y2 <-> APS Outputs/PhiE 3Y2
//     PlcTask Outputs/GVL_iXlinker.EtherCAT_Master_APSxxxx.Beckhoff_APS4xxx.Beckhoff_APS4xxxEK1122.A_0001_APS4322_7000_0017.APS_Comm_Outputs.CommControlWord <-> APS Comm Outputs/CommControlWord
//     PlcTask Outputs/GVL_iXlinker.EtherCAT_Master_APSxxxx.Beckhoff_APS4xxx.Beckhoff_APS4xxxEK1122.A_0001_APS4322_7000_0017.APS_Comm_Outputs.Data_1 <-> APS Comm Outputs/Data 1
//     PlcTask Inputs/GVL_iXlinker.EtherCAT_Master_APSxxxx.Beckhoff_APS4xxx.Beckhoff_APS4xxxEK1122.A_0001_APS4322_7000_0017.WcState.WcState <-> WcState/WcState
//     PlcTask Inputs/GVL_iXlinker.EtherCAT_Master_APSxxxx.Beckhoff_APS4xxx.Beckhoff_APS4xxxEK1122.A_0001_APS4322_7000_0017.WcState.InputToggle <-> WcState/InputToggle
//     PlcTask Inputs/GVL_iXlinker.EtherCAT_Master_APSxxxx.Beckhoff_APS4xxx.Beckhoff_APS4xxxEK1122.A_0001_APS4322_7000_0017.InfoData.AdsAddr <-> InfoData/AdsAddr
//     PlcTask Inputs/GVL_iXlinker.EtherCAT_Master_APSxxxx.Beckhoff_APS4xxx.Beckhoff_APS4xxxEK1122.A_0001_APS4322_7000_0017.InfoData.DcOutputShift <-> InfoData/DcOutputShift
//     PlcTask Inputs/GVL_iXlinker.EtherCAT_Master_APSxxxx.Beckhoff_APS4xxx.Beckhoff_APS4xxxEK1122.A_0001_APS4322_7000_0017.InfoData.DcInputShift <-> InfoData/DcInputShift
//     PlcTask Inputs/GVL_iXlinker.EtherCAT_Master_APSxxxx.Beckhoff_APS4xxx.Beckhoff_APS4xxxEK1122.A_0001_APS4322_7000_0017.InfoData.State <-> InfoData/State
//   PLC/PLC Instance <-> EtherCAT Master APSxxxx/Beckhoff APS4xxx/A_0002(APS4322-5000-0017)
//     PlcTask Inputs/GVL_iXlinker.EtherCAT_Master_APSxxxx.Beckhoff_APS4xxx.A_0002_APS4322_5000_0017.FB_Inputs.Status <-> FB Inputs/Status
//     PlcTask Inputs/GVL_iXlinker.EtherCAT_Master_APSxxxx.Beckhoff_APS4xxx.A_0002_APS4322_5000_0017.FB_Inputs.A0_X_Field <-> FB Inputs/A0 X-Field
//     PlcTask Inputs/GVL_iXlinker.EtherCAT_Master_APSxxxx.Beckhoff_APS4xxx.A_0002_APS4322_5000_0017.FB_Inputs.A2_X_Field <-> FB Inputs/A2 X-Field
//     PlcTask Inputs/GVL_iXlinker.EtherCAT_Master_APSxxxx.Beckhoff_APS4xxx.A_0002_APS4322_5000_0017.FB_Inputs.A4_X_Field <-> FB Inputs/A4 X-Field
//     PlcTask Inputs/GVL_iXlinker.EtherCAT_Master_APSxxxx.Beckhoff_APS4xxx.A_0002_APS4322_5000_0017.FB_Inputs.A6_X_Field <-> FB Inputs/A6 X-Field
//     PlcTask Inputs/GVL_iXlinker.EtherCAT_Master_APSxxxx.Beckhoff_APS4xxx.A_0002_APS4322_5000_0017.FB_Inputs.A8_X_Field <-> FB Inputs/A8 X-Field
//     PlcTask Inputs/GVL_iXlinker.EtherCAT_Master_APSxxxx.Beckhoff_APS4xxx.A_0002_APS4322_5000_0017.FB_Inputs.A0_Y_Field <-> FB Inputs/A0 Y-Field
//     PlcTask Inputs/GVL_iXlinker.EtherCAT_Master_APSxxxx.Beckhoff_APS4xxx.A_0002_APS4322_5000_0017.FB_Inputs.A2_Y_Field <-> FB Inputs/A2 Y-Field
//     PlcTask Inputs/GVL_iXlinker.EtherCAT_Master_APSxxxx.Beckhoff_APS4xxx.A_0002_APS4322_5000_0017.FB_Inputs.A4_Y_Field <-> FB Inputs/A4 Y-Field
//     PlcTask Inputs/GVL_iXlinker.EtherCAT_Master_APSxxxx.Beckhoff_APS4xxx.A_0002_APS4322_5000_0017.FB_Inputs.A6_Y_Field <-> FB Inputs/A6 Y-Field
//     PlcTask Inputs/GVL_iXlinker.EtherCAT_Master_APSxxxx.Beckhoff_APS4xxx.A_0002_APS4322_5000_0017.FB_Inputs.A8_Y_Field <-> FB Inputs/A8 Y-Field
//     PlcTask Inputs/GVL_iXlinker.EtherCAT_Master_APSxxxx.Beckhoff_APS4xxx.A_0002_APS4322_5000_0017.FB_Inputs.A0_Z_Field <-> FB Inputs/A0 Z-Field
//     PlcTask Inputs/GVL_iXlinker.EtherCAT_Master_APSxxxx.Beckhoff_APS4xxx.A_0002_APS4322_5000_0017.FB_Inputs.A2_Z_Field <-> FB Inputs/A2 Z-Field
//     PlcTask Inputs/GVL_iXlinker.EtherCAT_Master_APSxxxx.Beckhoff_APS4xxx.A_0002_APS4322_5000_0017.FB_Inputs.A4_Z_Field <-> FB Inputs/A4 Z-Field
//     PlcTask Inputs/GVL_iXlinker.EtherCAT_Master_APSxxxx.Beckhoff_APS4xxx.A_0002_APS4322_5000_0017.FB_Inputs.A6_Z_Field <-> FB Inputs/A6 Z-Field
//     PlcTask Inputs/GVL_iXlinker.EtherCAT_Master_APSxxxx.Beckhoff_APS4xxx.A_0002_APS4322_5000_0017.FB_Inputs.A8_Z_Field <-> FB Inputs/A8 Z-Field
//     PlcTask Inputs/GVL_iXlinker.EtherCAT_Master_APSxxxx.Beckhoff_APS4xxx.A_0002_APS4322_5000_0017.FB_Inputs.B1_X_Field <-> FB Inputs/B1 X-Field
//     PlcTask Inputs/GVL_iXlinker.EtherCAT_Master_APSxxxx.Beckhoff_APS4xxx.A_0002_APS4322_5000_0017.FB_Inputs.B3_X_Field <-> FB Inputs/B3 X-Field
//     PlcTask Inputs/GVL_iXlinker.EtherCAT_Master_APSxxxx.Beckhoff_APS4xxx.A_0002_APS4322_5000_0017.FB_Inputs.B5_X_Field <-> FB Inputs/B5 X-Field
//     PlcTask Inputs/GVL_iXlinker.EtherCAT_Master_APSxxxx.Beckhoff_APS4xxx.A_0002_APS4322_5000_0017.FB_Inputs.B7_X_Field <-> FB Inputs/B7 X-Field
//     PlcTask Inputs/GVL_iXlinker.EtherCAT_Master_APSxxxx.Beckhoff_APS4xxx.A_0002_APS4322_5000_0017.FB_Inputs.B9_X_Field <-> FB Inputs/B9 X-Field
//     PlcTask Inputs/GVL_iXlinker.EtherCAT_Master_APSxxxx.Beckhoff_APS4xxx.A_0002_APS4322_5000_0017.FB_Inputs.B1_Y_Field <-> FB Inputs/B1 Y-Field
//     PlcTask Inputs/GVL_iXlinker.EtherCAT_Master_APSxxxx.Beckhoff_APS4xxx.A_0002_APS4322_5000_0017.FB_Inputs.B3_Y_Field <-> FB Inputs/B3 Y-Field
//     PlcTask Inputs/GVL_iXlinker.EtherCAT_Master_APSxxxx.Beckhoff_APS4xxx.A_0002_APS4322_5000_0017.FB_Inputs.B5_Y_Field <-> FB Inputs/B5 Y-Field
//     PlcTask Inputs/GVL_iXlinker.EtherCAT_Master_APSxxxx.Beckhoff_APS4xxx.A_0002_APS4322_5000_0017.FB_Inputs.B7_Y_Field <-> FB Inputs/B7 Y-Field
//     PlcTask Inputs/GVL_iXlinker.EtherCAT_Master_APSxxxx.Beckhoff_APS4xxx.A_0002_APS4322_5000_0017.FB_Inputs.B9_Y_Field <-> FB Inputs/B9 Y-Field
//     PlcTask Inputs/GVL_iXlinker.EtherCAT_Master_APSxxxx.Beckhoff_APS4xxx.A_0002_APS4322_5000_0017.FB_Inputs.B1_Z_Field <-> FB Inputs/B1 Z-Field
//     PlcTask Inputs/GVL_iXlinker.EtherCAT_Master_APSxxxx.Beckhoff_APS4xxx.A_0002_APS4322_5000_0017.FB_Inputs.B3_Z_Field <-> FB Inputs/B3 Z-Field
//     PlcTask Inputs/GVL_iXlinker.EtherCAT_Master_APSxxxx.Beckhoff_APS4xxx.A_0002_APS4322_5000_0017.FB_Inputs.B5_Z_Field <-> FB Inputs/B5 Z-Field
//     PlcTask Inputs/GVL_iXlinker.EtherCAT_Master_APSxxxx.Beckhoff_APS4xxx.A_0002_APS4322_5000_0017.FB_Inputs.B7_Z_Field <-> FB Inputs/B7 Z-Field
//     PlcTask Inputs/GVL_iXlinker.EtherCAT_Master_APSxxxx.Beckhoff_APS4xxx.A_0002_APS4322_5000_0017.FB_Inputs.B9_Z_Field <-> FB Inputs/B9 Z-Field
//     PlcTask Inputs/GVL_iXlinker.EtherCAT_Master_APSxxxx.Beckhoff_APS4xxx.A_0002_APS4322_5000_0017.FB_Inputs.C0_X_Field <-> FB Inputs/C0 X-Field
//     PlcTask Inputs/GVL_iXlinker.EtherCAT_Master_APSxxxx.Beckhoff_APS4xxx.A_0002_APS4322_5000_0017.FB_Inputs.C2_X_Field <-> FB Inputs/C2 X-Field
//     PlcTask Inputs/GVL_iXlinker.EtherCAT_Master_APSxxxx.Beckhoff_APS4xxx.A_0002_APS4322_5000_0017.FB_Inputs.C4_X_Field <-> FB Inputs/C4 X-Field
//     PlcTask Inputs/GVL_iXlinker.EtherCAT_Master_APSxxxx.Beckhoff_APS4xxx.A_0002_APS4322_5000_0017.FB_Inputs.C6_X_Field <-> FB Inputs/C6 X-Field
//     PlcTask Inputs/GVL_iXlinker.EtherCAT_Master_APSxxxx.Beckhoff_APS4xxx.A_0002_APS4322_5000_0017.FB_Inputs.C8_X_Field <-> FB Inputs/C8 X-Field
//     PlcTask Inputs/GVL_iXlinker.EtherCAT_Master_APSxxxx.Beckhoff_APS4xxx.A_0002_APS4322_5000_0017.FB_Inputs.C0_Y_Field <-> FB Inputs/C0 Y-Field
//     PlcTask Inputs/GVL_iXlinker.EtherCAT_Master_APSxxxx.Beckhoff_APS4xxx.A_0002_APS4322_5000_0017.FB_Inputs.C2_Y_Field <-> FB Inputs/C2 Y-Field
//     PlcTask Inputs/GVL_iXlinker.EtherCAT_Master_APSxxxx.Beckhoff_APS4xxx.A_0002_APS4322_5000_0017.FB_Inputs.C4_Y_Field <-> FB Inputs/C4 Y-Field
//     PlcTask Inputs/GVL_iXlinker.EtherCAT_Master_APSxxxx.Beckhoff_APS4xxx.A_0002_APS4322_5000_0017.FB_Inputs.C6_Y_Field <-> FB Inputs/C6 Y-Field
//     PlcTask Inputs/GVL_iXlinker.EtherCAT_Master_APSxxxx.Beckhoff_APS4xxx.A_0002_APS4322_5000_0017.FB_Inputs.C8_Y_Field <-> FB Inputs/C8 Y-Field
//     PlcTask Inputs/GVL_iXlinker.EtherCAT_Master_APSxxxx.Beckhoff_APS4xxx.A_0002_APS4322_5000_0017.FB_Inputs.C0_Z_Field <-> FB Inputs/C0 Z-Field
//     PlcTask Inputs/GVL_iXlinker.EtherCAT_Master_APSxxxx.Beckhoff_APS4xxx.A_0002_APS4322_5000_0017.FB_Inputs.C2_Z_Field <-> FB Inputs/C2 Z-Field
//     PlcTask Inputs/GVL_iXlinker.EtherCAT_Master_APSxxxx.Beckhoff_APS4xxx.A_0002_APS4322_5000_0017.FB_Inputs.C4_Z_Field <-> FB Inputs/C4 Z-Field
//     PlcTask Inputs/GVL_iXlinker.EtherCAT_Master_APSxxxx.Beckhoff_APS4xxx.A_0002_APS4322_5000_0017.FB_Inputs.C6_Z_Field <-> FB Inputs/C6 Z-Field
//     PlcTask Inputs/GVL_iXlinker.EtherCAT_Master_APSxxxx.Beckhoff_APS4xxx.A_0002_APS4322_5000_0017.FB_Inputs.C8_Z_Field <-> FB Inputs/C8 Z-Field
//     PlcTask Inputs/GVL_iXlinker.EtherCAT_Master_APSxxxx.Beckhoff_APS4xxx.A_0002_APS4322_5000_0017.FB_Inputs.D1_X_Field <-> FB Inputs/D1 X-Field
//     PlcTask Inputs/GVL_iXlinker.EtherCAT_Master_APSxxxx.Beckhoff_APS4xxx.A_0002_APS4322_5000_0017.FB_Inputs.D3_X_Field <-> FB Inputs/D3 X-Field
//     PlcTask Inputs/GVL_iXlinker.EtherCAT_Master_APSxxxx.Beckhoff_APS4xxx.A_0002_APS4322_5000_0017.FB_Inputs.D5_X_Field <-> FB Inputs/D5 X-Field
//     PlcTask Inputs/GVL_iXlinker.EtherCAT_Master_APSxxxx.Beckhoff_APS4xxx.A_0002_APS4322_5000_0017.FB_Inputs.D7_X_Field <-> FB Inputs/D7 X-Field
//     PlcTask Inputs/GVL_iXlinker.EtherCAT_Master_APSxxxx.Beckhoff_APS4xxx.A_0002_APS4322_5000_0017.FB_Inputs.D9_X_Field <-> FB Inputs/D9 X-Field
//     PlcTask Inputs/GVL_iXlinker.EtherCAT_Master_APSxxxx.Beckhoff_APS4xxx.A_0002_APS4322_5000_0017.FB_Inputs.D1_Y_Field <-> FB Inputs/D1 Y-Field
//     PlcTask Inputs/GVL_iXlinker.EtherCAT_Master_APSxxxx.Beckhoff_APS4xxx.A_0002_APS4322_5000_0017.FB_Inputs.D3_Y_Field <-> FB Inputs/D3 Y-Field
//     PlcTask Inputs/GVL_iXlinker.EtherCAT_Master_APSxxxx.Beckhoff_APS4xxx.A_0002_APS4322_5000_0017.FB_Inputs.D5_Y_Field <-> FB Inputs/D5 Y-Field
//     PlcTask Inputs/GVL_iXlinker.EtherCAT_Master_APSxxxx.Beckhoff_APS4xxx.A_0002_APS4322_5000_0017.FB_Inputs.D7_Y_Field <-> FB Inputs/D7 Y-Field
//     PlcTask Inputs/GVL_iXlinker.EtherCAT_Master_APSxxxx.Beckhoff_APS4xxx.A_0002_APS4322_5000_0017.FB_Inputs.D9_Y_Field <-> FB Inputs/D9 Y-Field
//     PlcTask Inputs/GVL_iXlinker.EtherCAT_Master_APSxxxx.Beckhoff_APS4xxx.A_0002_APS4322_5000_0017.FB_Inputs.D1_Z_Field <-> FB Inputs/D1 Z-Field
//     PlcTask Inputs/GVL_iXlinker.EtherCAT_Master_APSxxxx.Beckhoff_APS4xxx.A_0002_APS4322_5000_0017.FB_Inputs.D3_Z_Field <-> FB Inputs/D3 Z-Field
//     PlcTask Inputs/GVL_iXlinker.EtherCAT_Master_APSxxxx.Beckhoff_APS4xxx.A_0002_APS4322_5000_0017.FB_Inputs.D5_Z_Field <-> FB Inputs/D5 Z-Field
//     PlcTask Inputs/GVL_iXlinker.EtherCAT_Master_APSxxxx.Beckhoff_APS4xxx.A_0002_APS4322_5000_0017.FB_Inputs.D7_Z_Field <-> FB Inputs/D7 Z-Field
//     PlcTask Inputs/GVL_iXlinker.EtherCAT_Master_APSxxxx.Beckhoff_APS4xxx.A_0002_APS4322_5000_0017.FB_Inputs.D9_Z_Field <-> FB Inputs/D9 Z-Field
//     PlcTask Inputs/GVL_iXlinker.EtherCAT_Master_APSxxxx.Beckhoff_APS4xxx.A_0002_APS4322_5000_0017.FB_Inputs.E0_X_Field <-> FB Inputs/E0 X-Field
//     PlcTask Inputs/GVL_iXlinker.EtherCAT_Master_APSxxxx.Beckhoff_APS4xxx.A_0002_APS4322_5000_0017.FB_Inputs.E2_X_Field <-> FB Inputs/E2 X-Field
//     PlcTask Inputs/GVL_iXlinker.EtherCAT_Master_APSxxxx.Beckhoff_APS4xxx.A_0002_APS4322_5000_0017.FB_Inputs.E4_X_Field <-> FB Inputs/E4 X-Field
//     PlcTask Inputs/GVL_iXlinker.EtherCAT_Master_APSxxxx.Beckhoff_APS4xxx.A_0002_APS4322_5000_0017.FB_Inputs.E6_X_Field <-> FB Inputs/E6 X-Field
//     PlcTask Inputs/GVL_iXlinker.EtherCAT_Master_APSxxxx.Beckhoff_APS4xxx.A_0002_APS4322_5000_0017.FB_Inputs.E8_X_Field <-> FB Inputs/E8 X-Field
//     PlcTask Inputs/GVL_iXlinker.EtherCAT_Master_APSxxxx.Beckhoff_APS4xxx.A_0002_APS4322_5000_0017.FB_Inputs.E0_Y_Field <-> FB Inputs/E0 Y-Field
//     PlcTask Inputs/GVL_iXlinker.EtherCAT_Master_APSxxxx.Beckhoff_APS4xxx.A_0002_APS4322_5000_0017.FB_Inputs.E2_Y_Field <-> FB Inputs/E2 Y-Field
//     PlcTask Inputs/GVL_iXlinker.EtherCAT_Master_APSxxxx.Beckhoff_APS4xxx.A_0002_APS4322_5000_0017.FB_Inputs.E4_Y_Field <-> FB Inputs/E4 Y-Field
//     PlcTask Inputs/GVL_iXlinker.EtherCAT_Master_APSxxxx.Beckhoff_APS4xxx.A_0002_APS4322_5000_0017.FB_Inputs.E6_Y_Field <-> FB Inputs/E6 Y-Field
//     PlcTask Inputs/GVL_iXlinker.EtherCAT_Master_APSxxxx.Beckhoff_APS4xxx.A_0002_APS4322_5000_0017.FB_Inputs.E8_Y_Field <-> FB Inputs/E8 Y-Field
//     PlcTask Inputs/GVL_iXlinker.EtherCAT_Master_APSxxxx.Beckhoff_APS4xxx.A_0002_APS4322_5000_0017.FB_Inputs.E0_Z_Field <-> FB Inputs/E0 Z-Field
//     PlcTask Inputs/GVL_iXlinker.EtherCAT_Master_APSxxxx.Beckhoff_APS4xxx.A_0002_APS4322_5000_0017.FB_Inputs.E2_Z_Field <-> FB Inputs/E2 Z-Field
//     PlcTask Inputs/GVL_iXlinker.EtherCAT_Master_APSxxxx.Beckhoff_APS4xxx.A_0002_APS4322_5000_0017.FB_Inputs.E4_Z_Field <-> FB Inputs/E4 Z-Field
//     PlcTask Inputs/GVL_iXlinker.EtherCAT_Master_APSxxxx.Beckhoff_APS4xxx.A_0002_APS4322_5000_0017.FB_Inputs.E6_Z_Field <-> FB Inputs/E6 Z-Field
//     PlcTask Inputs/GVL_iXlinker.EtherCAT_Master_APSxxxx.Beckhoff_APS4xxx.A_0002_APS4322_5000_0017.FB_Inputs.E8_Z_Field <-> FB Inputs/E8 Z-Field
//     PlcTask Inputs/GVL_iXlinker.EtherCAT_Master_APSxxxx.Beckhoff_APS4xxx.A_0002_APS4322_5000_0017.FB_Inputs.F1_X_Field <-> FB Inputs/F1 X-Field
//     PlcTask Inputs/GVL_iXlinker.EtherCAT_Master_APSxxxx.Beckhoff_APS4xxx.A_0002_APS4322_5000_0017.FB_Inputs.F3_X_Field <-> FB Inputs/F3 X-Field
//     PlcTask Inputs/GVL_iXlinker.EtherCAT_Master_APSxxxx.Beckhoff_APS4xxx.A_0002_APS4322_5000_0017.FB_Inputs.F5_X_Field <-> FB Inputs/F5 X-Field
//     PlcTask Inputs/GVL_iXlinker.EtherCAT_Master_APSxxxx.Beckhoff_APS4xxx.A_0002_APS4322_5000_0017.FB_Inputs.F7_X_Field <-> FB Inputs/F7 X-Field
//     PlcTask Inputs/GVL_iXlinker.EtherCAT_Master_APSxxxx.Beckhoff_APS4xxx.A_0002_APS4322_5000_0017.FB_Inputs.F9_X_Field <-> FB Inputs/F9 X-Field
//     PlcTask Inputs/GVL_iXlinker.EtherCAT_Master_APSxxxx.Beckhoff_APS4xxx.A_0002_APS4322_5000_0017.FB_Inputs.F1_Y_Field <-> FB Inputs/F1 Y-Field
//     PlcTask Inputs/GVL_iXlinker.EtherCAT_Master_APSxxxx.Beckhoff_APS4xxx.A_0002_APS4322_5000_0017.FB_Inputs.F3_Y_Field <-> FB Inputs/F3 Y-Field
//     PlcTask Inputs/GVL_iXlinker.EtherCAT_Master_APSxxxx.Beckhoff_APS4xxx.A_0002_APS4322_5000_0017.FB_Inputs.F5_Y_Field <-> FB Inputs/F5 Y-Field
//     PlcTask Inputs/GVL_iXlinker.EtherCAT_Master_APSxxxx.Beckhoff_APS4xxx.A_0002_APS4322_5000_0017.FB_Inputs.F7_Y_Field <-> FB Inputs/F7 Y-Field
//     PlcTask Inputs/GVL_iXlinker.EtherCAT_Master_APSxxxx.Beckhoff_APS4xxx.A_0002_APS4322_5000_0017.FB_Inputs.F9_Y_Field <-> FB Inputs/F9 Y-Field
//     PlcTask Inputs/GVL_iXlinker.EtherCAT_Master_APSxxxx.Beckhoff_APS4xxx.A_0002_APS4322_5000_0017.FB_Inputs.F1_Z_Field <-> FB Inputs/F1 Z-Field
//     PlcTask Inputs/GVL_iXlinker.EtherCAT_Master_APSxxxx.Beckhoff_APS4xxx.A_0002_APS4322_5000_0017.FB_Inputs.F3_Z_Field <-> FB Inputs/F3 Z-Field
//     PlcTask Inputs/GVL_iXlinker.EtherCAT_Master_APSxxxx.Beckhoff_APS4xxx.A_0002_APS4322_5000_0017.FB_Inputs.F5_Z_Field <-> FB Inputs/F5 Z-Field
//     PlcTask Inputs/GVL_iXlinker.EtherCAT_Master_APSxxxx.Beckhoff_APS4xxx.A_0002_APS4322_5000_0017.FB_Inputs.F7_Z_Field <-> FB Inputs/F7 Z-Field
//     PlcTask Inputs/GVL_iXlinker.EtherCAT_Master_APSxxxx.Beckhoff_APS4xxx.A_0002_APS4322_5000_0017.FB_Inputs.F9_Z_Field <-> FB Inputs/F9 Z-Field
//     PlcTask Inputs/GVL_iXlinker.EtherCAT_Master_APSxxxx.Beckhoff_APS4xxx.A_0002_APS4322_5000_0017.FB_Inputs.G0_X_Field <-> FB Inputs/G0 X-Field
//     PlcTask Inputs/GVL_iXlinker.EtherCAT_Master_APSxxxx.Beckhoff_APS4xxx.A_0002_APS4322_5000_0017.FB_Inputs.G2_X_Field <-> FB Inputs/G2 X-Field
//     PlcTask Inputs/GVL_iXlinker.EtherCAT_Master_APSxxxx.Beckhoff_APS4xxx.A_0002_APS4322_5000_0017.FB_Inputs.G4_X_Field <-> FB Inputs/G4 X-Field
//     PlcTask Inputs/GVL_iXlinker.EtherCAT_Master_APSxxxx.Beckhoff_APS4xxx.A_0002_APS4322_5000_0017.FB_Inputs.G6_X_Field <-> FB Inputs/G6 X-Field
//     PlcTask Inputs/GVL_iXlinker.EtherCAT_Master_APSxxxx.Beckhoff_APS4xxx.A_0002_APS4322_5000_0017.FB_Inputs.G8_X_Field <-> FB Inputs/G8 X-Field
//     PlcTask Inputs/GVL_iXlinker.EtherCAT_Master_APSxxxx.Beckhoff_APS4xxx.A_0002_APS4322_5000_0017.FB_Inputs.G0_Y_Field <-> FB Inputs/G0 Y-Field
//     PlcTask Inputs/GVL_iXlinker.EtherCAT_Master_APSxxxx.Beckhoff_APS4xxx.A_0002_APS4322_5000_0017.FB_Inputs.G2_Y_Field <-> FB Inputs/G2 Y-Field
//     PlcTask Inputs/GVL_iXlinker.EtherCAT_Master_APSxxxx.Beckhoff_APS4xxx.A_0002_APS4322_5000_0017.FB_Inputs.G4_Y_Field <-> FB Inputs/G4 Y-Field
//     PlcTask Inputs/GVL_iXlinker.EtherCAT_Master_APSxxxx.Beckhoff_APS4xxx.A_0002_APS4322_5000_0017.FB_Inputs.G6_Y_Field <-> FB Inputs/G6 Y-Field
//     PlcTask Inputs/GVL_iXlinker.EtherCAT_Master_APSxxxx.Beckhoff_APS4xxx.A_0002_APS4322_5000_0017.FB_Inputs.G8_Y_Field <-> FB Inputs/G8 Y-Field
//     PlcTask Inputs/GVL_iXlinker.EtherCAT_Master_APSxxxx.Beckhoff_APS4xxx.A_0002_APS4322_5000_0017.FB_Inputs.G0_Z_Field <-> FB Inputs/G0 Z-Field
//     PlcTask Inputs/GVL_iXlinker.EtherCAT_Master_APSxxxx.Beckhoff_APS4xxx.A_0002_APS4322_5000_0017.FB_Inputs.G2_Z_Field <-> FB Inputs/G2 Z-Field
//     PlcTask Inputs/GVL_iXlinker.EtherCAT_Master_APSxxxx.Beckhoff_APS4xxx.A_0002_APS4322_5000_0017.FB_Inputs.G4_Z_Field <-> FB Inputs/G4 Z-Field
//     PlcTask Inputs/GVL_iXlinker.EtherCAT_Master_APSxxxx.Beckhoff_APS4xxx.A_0002_APS4322_5000_0017.FB_Inputs.G6_Z_Field <-> FB Inputs/G6 Z-Field
//     PlcTask Inputs/GVL_iXlinker.EtherCAT_Master_APSxxxx.Beckhoff_APS4xxx.A_0002_APS4322_5000_0017.FB_Inputs.G8_Z_Field <-> FB Inputs/G8 Z-Field
//     PlcTask Inputs/GVL_iXlinker.EtherCAT_Master_APSxxxx.Beckhoff_APS4xxx.A_0002_APS4322_5000_0017.FB_Inputs.H1_X_Field <-> FB Inputs/H1 X-Field
//     PlcTask Inputs/GVL_iXlinker.EtherCAT_Master_APSxxxx.Beckhoff_APS4xxx.A_0002_APS4322_5000_0017.FB_Inputs.H3_X_Field <-> FB Inputs/H3 X-Field
//     PlcTask Inputs/GVL_iXlinker.EtherCAT_Master_APSxxxx.Beckhoff_APS4xxx.A_0002_APS4322_5000_0017.FB_Inputs.H5_X_Field <-> FB Inputs/H5 X-Field
//     PlcTask Inputs/GVL_iXlinker.EtherCAT_Master_APSxxxx.Beckhoff_APS4xxx.A_0002_APS4322_5000_0017.FB_Inputs.H7_X_Field <-> FB Inputs/H7 X-Field
//     PlcTask Inputs/GVL_iXlinker.EtherCAT_Master_APSxxxx.Beckhoff_APS4xxx.A_0002_APS4322_5000_0017.FB_Inputs.H9_X_Field <-> FB Inputs/H9 X-Field
//     PlcTask Inputs/GVL_iXlinker.EtherCAT_Master_APSxxxx.Beckhoff_APS4xxx.A_0002_APS4322_5000_0017.FB_Inputs.H1_Y_Field <-> FB Inputs/H1 Y-Field
//     PlcTask Inputs/GVL_iXlinker.EtherCAT_Master_APSxxxx.Beckhoff_APS4xxx.A_0002_APS4322_5000_0017.FB_Inputs.H3_Y_Field <-> FB Inputs/H3 Y-Field
//     PlcTask Inputs/GVL_iXlinker.EtherCAT_Master_APSxxxx.Beckhoff_APS4xxx.A_0002_APS4322_5000_0017.FB_Inputs.H5_Y_Field <-> FB Inputs/H5 Y-Field
//     PlcTask Inputs/GVL_iXlinker.EtherCAT_Master_APSxxxx.Beckhoff_APS4xxx.A_0002_APS4322_5000_0017.FB_Inputs.H7_Y_Field <-> FB Inputs/H7 Y-Field
//     PlcTask Inputs/GVL_iXlinker.EtherCAT_Master_APSxxxx.Beckhoff_APS4xxx.A_0002_APS4322_5000_0017.FB_Inputs.H9_Y_Field <-> FB Inputs/H9 Y-Field
//     PlcTask Inputs/GVL_iXlinker.EtherCAT_Master_APSxxxx.Beckhoff_APS4xxx.A_0002_APS4322_5000_0017.FB_Inputs.H1_Z_Field <-> FB Inputs/H1 Z-Field
//     PlcTask Inputs/GVL_iXlinker.EtherCAT_Master_APSxxxx.Beckhoff_APS4xxx.A_0002_APS4322_5000_0017.FB_Inputs.H3_Z_Field <-> FB Inputs/H3 Z-Field
//     PlcTask Inputs/GVL_iXlinker.EtherCAT_Master_APSxxxx.Beckhoff_APS4xxx.A_0002_APS4322_5000_0017.FB_Inputs.H5_Z_Field <-> FB Inputs/H5 Z-Field
//     PlcTask Inputs/GVL_iXlinker.EtherCAT_Master_APSxxxx.Beckhoff_APS4xxx.A_0002_APS4322_5000_0017.FB_Inputs.H7_Z_Field <-> FB Inputs/H7 Z-Field
//     PlcTask Inputs/GVL_iXlinker.EtherCAT_Master_APSxxxx.Beckhoff_APS4xxx.A_0002_APS4322_5000_0017.FB_Inputs.H9_Z_Field <-> FB Inputs/H9 Z-Field
//     PlcTask Inputs/GVL_iXlinker.EtherCAT_Master_APSxxxx.Beckhoff_APS4xxx.A_0002_APS4322_5000_0017.FB_Inputs.I0_X_Field <-> FB Inputs/I0 X-Field
//     PlcTask Inputs/GVL_iXlinker.EtherCAT_Master_APSxxxx.Beckhoff_APS4xxx.A_0002_APS4322_5000_0017.FB_Inputs.I2_X_Field <-> FB Inputs/I2 X-Field
//     PlcTask Inputs/GVL_iXlinker.EtherCAT_Master_APSxxxx.Beckhoff_APS4xxx.A_0002_APS4322_5000_0017.FB_Inputs.I4_X_Field <-> FB Inputs/I4 X-Field
//     PlcTask Inputs/GVL_iXlinker.EtherCAT_Master_APSxxxx.Beckhoff_APS4xxx.A_0002_APS4322_5000_0017.FB_Inputs.I6_X_Field <-> FB Inputs/I6 X-Field
//     PlcTask Inputs/GVL_iXlinker.EtherCAT_Master_APSxxxx.Beckhoff_APS4xxx.A_0002_APS4322_5000_0017.FB_Inputs.I8_X_Field <-> FB Inputs/I8 X-Field
//     PlcTask Inputs/GVL_iXlinker.EtherCAT_Master_APSxxxx.Beckhoff_APS4xxx.A_0002_APS4322_5000_0017.FB_Inputs.I0_Y_Field <-> FB Inputs/I0 Y-Field
//     PlcTask Inputs/GVL_iXlinker.EtherCAT_Master_APSxxxx.Beckhoff_APS4xxx.A_0002_APS4322_5000_0017.FB_Inputs.I2_Y_Field <-> FB Inputs/I2 Y-Field
//     PlcTask Inputs/GVL_iXlinker.EtherCAT_Master_APSxxxx.Beckhoff_APS4xxx.A_0002_APS4322_5000_0017.FB_Inputs.I4_Y_Field <-> FB Inputs/I4 Y-Field
//     PlcTask Inputs/GVL_iXlinker.EtherCAT_Master_APSxxxx.Beckhoff_APS4xxx.A_0002_APS4322_5000_0017.FB_Inputs.I6_Y_Field <-> FB Inputs/I6 Y-Field
//     PlcTask Inputs/GVL_iXlinker.EtherCAT_Master_APSxxxx.Beckhoff_APS4xxx.A_0002_APS4322_5000_0017.FB_Inputs.I8_Y_Field <-> FB Inputs/I8 Y-Field
//     PlcTask Inputs/GVL_iXlinker.EtherCAT_Master_APSxxxx.Beckhoff_APS4xxx.A_0002_APS4322_5000_0017.FB_Inputs.I0_Z_Field <-> FB Inputs/I0 Z-Field
//     PlcTask Inputs/GVL_iXlinker.EtherCAT_Master_APSxxxx.Beckhoff_APS4xxx.A_0002_APS4322_5000_0017.FB_Inputs.I2_Z_Field <-> FB Inputs/I2 Z-Field
//     PlcTask Inputs/GVL_iXlinker.EtherCAT_Master_APSxxxx.Beckhoff_APS4xxx.A_0002_APS4322_5000_0017.FB_Inputs.I4_Z_Field <-> FB Inputs/I4 Z-Field
//     PlcTask Inputs/GVL_iXlinker.EtherCAT_Master_APSxxxx.Beckhoff_APS4xxx.A_0002_APS4322_5000_0017.FB_Inputs.I6_Z_Field <-> FB Inputs/I6 Z-Field
//     PlcTask Inputs/GVL_iXlinker.EtherCAT_Master_APSxxxx.Beckhoff_APS4xxx.A_0002_APS4322_5000_0017.FB_Inputs.I8_Z_Field <-> FB Inputs/I8 Z-Field
//     PlcTask Inputs/GVL_iXlinker.EtherCAT_Master_APSxxxx.Beckhoff_APS4xxx.A_0002_APS4322_5000_0017.FB_Inputs.J1_X_Field <-> FB Inputs/J1 X-Field
//     PlcTask Inputs/GVL_iXlinker.EtherCAT_Master_APSxxxx.Beckhoff_APS4xxx.A_0002_APS4322_5000_0017.FB_Inputs.J3_X_Field <-> FB Inputs/J3 X-Field
//     PlcTask Inputs/GVL_iXlinker.EtherCAT_Master_APSxxxx.Beckhoff_APS4xxx.A_0002_APS4322_5000_0017.FB_Inputs.J5_X_Field <-> FB Inputs/J5 X-Field
//     PlcTask Inputs/GVL_iXlinker.EtherCAT_Master_APSxxxx.Beckhoff_APS4xxx.A_0002_APS4322_5000_0017.FB_Inputs.J7_X_Field <-> FB Inputs/J7 X-Field
//     PlcTask Inputs/GVL_iXlinker.EtherCAT_Master_APSxxxx.Beckhoff_APS4xxx.A_0002_APS4322_5000_0017.FB_Inputs.J9_X_Field <-> FB Inputs/J9 X-Field
//     PlcTask Inputs/GVL_iXlinker.EtherCAT_Master_APSxxxx.Beckhoff_APS4xxx.A_0002_APS4322_5000_0017.FB_Inputs.J1_Y_Field <-> FB Inputs/J1 Y-Field
//     PlcTask Inputs/GVL_iXlinker.EtherCAT_Master_APSxxxx.Beckhoff_APS4xxx.A_0002_APS4322_5000_0017.FB_Inputs.J3_Y_Field <-> FB Inputs/J3 Y-Field
//     PlcTask Inputs/GVL_iXlinker.EtherCAT_Master_APSxxxx.Beckhoff_APS4xxx.A_0002_APS4322_5000_0017.FB_Inputs.J5_Y_Field <-> FB Inputs/J5 Y-Field
//     PlcTask Inputs/GVL_iXlinker.EtherCAT_Master_APSxxxx.Beckhoff_APS4xxx.A_0002_APS4322_5000_0017.FB_Inputs.J7_Y_Field <-> FB Inputs/J7 Y-Field
//     PlcTask Inputs/GVL_iXlinker.EtherCAT_Master_APSxxxx.Beckhoff_APS4xxx.A_0002_APS4322_5000_0017.FB_Inputs.J9_Y_Field <-> FB Inputs/J9 Y-Field
//     PlcTask Inputs/GVL_iXlinker.EtherCAT_Master_APSxxxx.Beckhoff_APS4xxx.A_0002_APS4322_5000_0017.FB_Inputs.J1_Z_Field <-> FB Inputs/J1 Z-Field
//     PlcTask Inputs/GVL_iXlinker.EtherCAT_Master_APSxxxx.Beckhoff_APS4xxx.A_0002_APS4322_5000_0017.FB_Inputs.J3_Z_Field <-> FB Inputs/J3 Z-Field
//     PlcTask Inputs/GVL_iXlinker.EtherCAT_Master_APSxxxx.Beckhoff_APS4xxx.A_0002_APS4322_5000_0017.FB_Inputs.J5_Z_Field <-> FB Inputs/J5 Z-Field
//     PlcTask Inputs/GVL_iXlinker.EtherCAT_Master_APSxxxx.Beckhoff_APS4xxx.A_0002_APS4322_5000_0017.FB_Inputs.J7_Z_Field <-> FB Inputs/J7 Z-Field
//     PlcTask Inputs/GVL_iXlinker.EtherCAT_Master_APSxxxx.Beckhoff_APS4xxx.A_0002_APS4322_5000_0017.FB_Inputs.J9_Z_Field <-> FB Inputs/J9 Z-Field
//     PlcTask Inputs/GVL_iXlinker.EtherCAT_Master_APSxxxx.Beckhoff_APS4xxx.A_0002_APS4322_5000_0017.WcState.WcState <-> WcState/WcState
//     PlcTask Inputs/GVL_iXlinker.EtherCAT_Master_APSxxxx.Beckhoff_APS4xxx.A_0002_APS4322_5000_0017.WcState.InputToggle <-> WcState/InputToggle
//     PlcTask Inputs/GVL_iXlinker.EtherCAT_Master_APSxxxx.Beckhoff_APS4xxx.A_0002_APS4322_5000_0017.InfoData.DcOutputShift <-> InfoData/DcOutputShift
//     PlcTask Inputs/GVL_iXlinker.EtherCAT_Master_APSxxxx.Beckhoff_APS4xxx.A_0002_APS4322_5000_0017.InfoData.DcInputShift <-> InfoData/DcInputShift
//     PlcTask Inputs/GVL_iXlinker.EtherCAT_Master_APSxxxx.Beckhoff_APS4xxx.A_0002_APS4322_5000_0017.InfoData.State <-> InfoData/State
//   PLC/PLC Instance <-> EtherCAT_Master_APSxxxx
//     PlcTask Inputs/GVL_iXlinker.EtherCAT_Master_APSxxxx.SyncUnits._default._unreferenced.WcState.WcState <-> SyncUnits/<default>/<unreferenced>/WcState/WcState
//     PlcTask Inputs/GVL_iXlinker.EtherCAT_Master_APSxxxx.SyncUnits._default._unreferenced.InfoData.ObjectId <-> SyncUnits/<default>/<unreferenced>/InfoData/ObjectId
//     PlcTask Inputs/GVL_iXlinker.EtherCAT_Master_APSxxxx.SyncUnits._default._unreferenced.InfoData.State <-> SyncUnits/<default>/<unreferenced>/InfoData/State
//     PlcTask Inputs/GVL_iXlinker.EtherCAT_Master_APSxxxx.SyncUnits._default._unreferenced.InfoData.SlaveCount <-> SyncUnits/<default>/<unreferenced>/InfoData/SlaveCount
//     PlcTask Inputs/GVL_iXlinker.EtherCAT_Master_APSxxxx.SyncUnits._default.PlcTask.WcState.WcState <-> SyncUnits/<default>/PlcTask/WcState/WcState
//     PlcTask Inputs/GVL_iXlinker.EtherCAT_Master_APSxxxx.SyncUnits._default.PlcTask.InfoData.ObjectId <-> SyncUnits/<default>/PlcTask/InfoData/ObjectId
//     PlcTask Inputs/GVL_iXlinker.EtherCAT_Master_APSxxxx.SyncUnits._default.PlcTask.InfoData.State <-> SyncUnits/<default>/PlcTask/InfoData/State
//     PlcTask Inputs/GVL_iXlinker.EtherCAT_Master_APSxxxx.SyncUnits._default.PlcTask.InfoData.SlaveCount <-> SyncUnits/<default>/PlcTask/InfoData/SlaveCount
//     PlcTask Inputs/GVL_iXlinker.EtherCAT_Master_APSxxxx.Inputs.SlaveCount <-> Inputs/SlaveCount
//     PlcTask Inputs/GVL_iXlinker.EtherCAT_Master_APSxxxx.Inputs.DevState <-> Inputs/DevState
//     PlcTask Inputs/GVL_iXlinker.EtherCAT_Master_APSxxxx.Inputs.Frm{0..25}State <-> Inputs/Frm{0..25}State  (26 links)
//     PlcTask Inputs/GVL_iXlinker.EtherCAT_Master_APSxxxx.Inputs.Frm{0..25}WcState <-> Inputs/Frm{0..25}WcState  (26 links)
//     PlcTask Inputs/GVL_iXlinker.EtherCAT_Master_APSxxxx.Inputs.Frm{0..25}InputToggle <-> Inputs/Frm{0..25}InputToggle  (26 links)
//     PlcTask Outputs/GVL_iXlinker.EtherCAT_Master_APSxxxx.Outputs.DevCtrl <-> Outputs/DevCtrl
//     PlcTask Outputs/GVL_iXlinker.EtherCAT_Master_APSxxxx.Outputs.Frm{0..25}Ctrl <-> Outputs/Frm{0..25}Ctrl  (26 links)
//     PlcTask Outputs/GVL_iXlinker.EtherCAT_Master_APSxxxx.Outputs.Frm{0..25}WcCtrl <-> Outputs/Frm{0..25}WcCtrl  (26 links)
//     PlcTask Inputs/GVL_iXlinker.EtherCAT_Master_APSxxxx.InfoData.ChangeCount <-> InfoData/ChangeCount
//     PlcTask Inputs/GVL_iXlinker.EtherCAT_Master_APSxxxx.InfoData.DevId <-> InfoData/DevId
//     PlcTask Inputs/GVL_iXlinker.EtherCAT_Master_APSxxxx.InfoData.AmsNetId <-> InfoData/AmsNetId
//     PlcTask Inputs/GVL_iXlinker.EtherCAT_Master_APSxxxx.InfoData.CfgSlaveCount <-> InfoData/CfgSlaveCount
//     PlcTask Inputs/GVL_iXlinker.EtherCAT_Master_APSxxxx.InfoData.DcToTcTimeOffset <-> InfoData/DcToTcTimeOffset
//     PlcTask Inputs/GVL_iXlinker.EtherCAT_Master_APSxxxx.InfoData.DcToExtTimeOffset <-> InfoData/DcToExtTimeOffset

CONFIGURATION PLC
    RESOURCE PLC ON TwinCAT3
        TASK PlcTask(INTERVAL := T#10ms, PRIORITY := 20);
        PROGRAM MAIN WITH PlcTask : MAIN;
    END_RESOURCE
END_CONFIGURATION

